(* Logix 5000 project; controller cal1632 1756-L62 rev 16.20; software revision 16.05; part 3 of 57 *)
(* tags used below, declared in another part *)
   AFI : BOOL;
   FAULT : BOOL;
   HMI : BOOL;
   p01_dint_to_hmi : DINT[16];
   p01_param_heater_hl : REAL;
   p01_param_process_air_hl : REAL;
   p01_param_process_air_max : REAL;
   p01_param_temp_limit : REAL;
   p01r01 : routine;
   p01r02 : routine;
   p01r02_all_fans_stopped : BOOL;
   p01r02_batch_run_time : DINT;
   p01r02_batch_run_time_hrs : DINT;
   p01r02_ethernet_comm : DINT;
   p01r02_fault_exists : BOOL;
   p01r02_flash_bit : BOOL;
   p01r02_flash_timer_off : TIMER;
   p01r02_flash_timer_on : TIMER;
   p01r02_plc_faults : DINT;
   p01r02_plc_scan_time : DINT;
   p01r02_plc_scan_time_in_sec : REAL;
   p01r02_timer_batch : TIMER;
   p01r02_timer_fault : TIMER[25];
   p01r02_timer_half_second_off : TIMER;
   p01r02_timer_half_second_on : TIMER;
   p01r02_timer_second : TIMER[2];
   p01r02_timer_warning : TIMER[4];
   p01r02_unack_fault : BOOL;
   p01r02_unack_warning : BOOL;
   p01r02_vfd_comm_2 : DINT[50];
   p01r02_warnings_exists : BOOL;
   p01r03 : routine;
   p01r04 : routine;
   p01r05 : routine;
   p01r06 : routine;
   p01r07 : routine;
   p01r08 : routine;
   p01r09 : routine;
   p01r09_pb_global_reset : BOOL;
   p01r10 : routine;
   p01r11 : routine;
   p01r12 : routine;
   p01r13 : routine;
   p01r13_line_running : BOOL;
   p02_dint_from_hmi : hmi_dint;
   p11r31_request_auto_run : BOOL;
   p11r32_request_auto_run : BOOL;
   p12r31_request_auto_run : BOOL;
   p12r32_request_auto_run : BOOL;
   p13r31_request_auto_run : BOOL;
   p13r32_request_auto_run : BOOL;
   p23_do_enable_impreg_exhaust_fan : BOOL;
   p23r13_request_auto_run : BOOL;

   p26r04_ulb_prs_scp : SYS_SCP := (Input := -85.5, Input_Min := 3.5, Input_Max := 20.0, Output_Min := 5397.0, Output_Max := 30840.0, Output := 5397.0);
   p26r05 : routine := (comment := -1073741761);
   p26r05_timer_fault : TIMER[4];
   p26r05_timer_warning : TIMER[4];
   p26r06 : routine := (comment := -1073741572);
   p26r06_timer_fault : TIMER[4];
   p26r06_timer_warning : TIMER[4];
   p26r07 : routine := (comment := -1073741761);
   p26r07_timer_fault : TIMER[4];
   p26r07_timer_warning : TIMER[4];
   p26r08 : routine := (comment := -1073741761);
   p26r08_timer_fault : TIMER[4];
   p26r08_timer_warning : TIMER[4];
   p26r09 : routine := (comment := -1073741761);
   p26r09_timer_fault : TIMER[4];
   p26r09_timer_warning : TIMER[4];
   p26r10 : routine := (comment := -1073741777);
   p26r10_timer_fault : TIMER[4];
   p26r10_timer_warning : TIMER[4];
   p26r10_ula_selected_tension : REAL := 3.0;
   p26r10_ulb_selected_tension : REAL := 3.0;
   p26r10_unwind_a_brake_torque : REAL := -9.417255;
   p26r10_unwind_a_dia_ft : REAL := -6.2809243;
   p26r10_unwind_b_brake_torque : REAL := -10.6875;
   p26r10_unwind_b_dia_ft : REAL := -7.125;
   p27_ao_dia_a : REAL := -38.8816;
   p27_ao_dia_b : REAL := 8.07605;
   p27_dint_to_hmi : DINT[16] := ([0] := 4);
   p27_inactive_tension_sp : REAL;
   p27_lft_a_prs_input_max : REAL := 30959.0;
   p27_lft_a_prs_input_min : REAL := 200.0;
   p27_lft_a_prs_output_max : REAL := 55.0;
   p27_lft_a_prs_output_min : REAL := 4.0;
   p27_lft_b_prs_input_max : REAL := 30959.0;
   p27_lft_b_prs_input_min : REAL := 60.0;
   p27_lft_b_prs_output_max : REAL := 55.0;
   p27_lft_b_prs_output_min : REAL := 4.0;
   p27_lla_prs_input_max : REAL := 20.0;
   p27_lla_prs_input_min : REAL := 3.5;
   p27_lla_prs_output_max : REAL := 30840.0;
   p27_lla_prs_output_min : REAL := 5397.0;
   p27_lla_prs_scp : SYS_SCP := (Input := -38.914757, Input_Min := 3.5, Input_Max := 20.0, Output_Min := 5397.0, Output_Max := 30840.0, Output := 5397.0);
   p27_llb_prs_input_max : REAL := 20.0;
   p27_llb_prs_input_min : REAL := 3.5;
   p27_llb_prs_output_max : REAL := 30840.0;
   p27_llb_prs_output_min : REAL := 5397.0;
   p27_llb_prs_scp : SYS_SCP := (Input := 8.07605, Input_Min := 3.5, Input_Max := 20.0, Output_Min := 5397.0, Output_Max := 30840.0, Output := 12453.269);
   p27_real_to_hmi : REAL[112] := ([0] := -38.8816, [1] := 8.043039);
   p27r01 : routine := (comment := 7);
   p27r02 : routine := (comment := -1073741761);
   p27r02_fault_exists : BOOL;
   p27r02_timer_fault : TIMER[4];
   p27r02_timer_warning : TIMER[4];
   p27r02_unack_fault : BOOL;
   p27r02_unack_warning : BOOL;
   p27r02_warning_exists : BOOL;
   p27r03 : routine := (comment := -1073741761);
   p27r03_a_radius : REAL := -19.4408;
   p27r03_ai_dia_a_sensor : REAL := 43.9408;
   p27r03_ai_dia_b_sensor : REAL := 8.0619755;
   p27r03_b_radius : REAL := 4.038025;
   p27r03_lower_A_tension_on : BOOL;
   p27r03_lower_B_tension_on : BOOL := 1;
   p27r03_ltf_a_diameter_scp : SYS_SCP := (Input := 24279.0, Input_Min := 200.0, Input_Max := 30959.0, Output_Min := 4.0, Output_Max := 55.0, Output := 43.924217);
   p27r03_ltf_b_diameter_scp : SYS_SCP := (Input := 2521.0, Input_Min := 60.0, Input_Max := 30959.0, Output_Min := 4.0, Output_Max := 55.0, Output := 8.0619755);
   p27r03_timer_fault : TIMER[4];
   p27r03_timer_warning : TIMER[4];
   p27r03_winder_a_distance : REAL := 24.5;
   p27r03_winder_b_distance : REAL := 12.1;
   p27r04 : routine := (comment := -1073741761);
   p27r04_timer_fault : TIMER[4];
   p27r04_timer_warning : TIMER[4];
   p27r05 : routine := (comment := -1073741761);
   p27r05_lla_mode_tension : BOOL;
   p27r05_llb_mode_tension : BOOL := 1;
   p27r05_timer_fault : TIMER[4];
   p27r05_timer_warning : TIMER[4];
   p27r06 : routine := (comment := -1073741572);
   p27r06_timer_fault : TIMER[4];
   p27r06_timer_warning : TIMER[4];
   p27r07 : routine := (comment := -1073741761);
   p27r07_timer_fault : TIMER[4];
   p27r07_timer_warning : TIMER[4];
   p27r08 : routine := (comment := -1073741761);
   p27r08_timer_fault : TIMER[4];
   p27r08_timer_warning : TIMER[4];
   p27r09 : routine := (comment := -1073741761);
   p27r09_a_enable_toggle : SYS_Toggle;
   p27r09_b_enable_toggle : SYS_Toggle := (toggle_state := 1);
   p27r09_timer_fault : TIMER[4];
   p27r09_timer_warning : TIMER[4];
   p27r10 : routine := (comment := -1073741777);
   p27r10_lla_selected_tension : REAL;
   p27r10_llb_selected_tension : REAL := 3.0;
   p27r10_timer_fault : TIMER[4];
   p27r10_timer_warning : TIMER[4];
   p27r10_unwind_a_brake_torque : REAL;
   p27r10_unwind_a_dia_ft : REAL := -3.2428963;
   p27r10_unwind_b_brake_torque : REAL := 1.0095062;
   p27r10_unwind_b_dia_ft : REAL := 0.67300415;
   p27r11 : routine;
   p289_di_ss_jog : BOOL;
   p289_di_ss_run : BOOL;
   p28_ai_slitter_amps : REAL;
   p28_ai_slitter_hz : REAL := -3.8146973e-06;
   p28_ai_slitter_speed : REAL;
   p28_ao_sltr_selected_speed : REAL;
   p28_di_brake : BOOL := 1;
   p28_di_motor : BOOL := 1;
   p28_di_slitter : acs800_di_normal;
   p28_dint_to_hmi : DINT[16] := ([0] := 4, [1] := 1024);
   p28_do_slt_air_supply_sv : BOOL;
   p28_do_sltr : acs800_do_normal;
   p28_real_to_hmi : REAL[112] := ([7] := -3.8146973e-06);
   p28_slitter_on : SYS_Toggle;
   p28r01 : routine := (comment := 7);
   p28r02 : routine := (comment := -1073741761);
   p28r02_fault_exists : BOOL;
   p28r02_timer_fault : TIMER[4];
   p28r02_timer_warning : TIMER[4];
   p28r02_unack_fault : BOOL;
   p28r02_unack_warning : BOOL;
   p28r02_warning_exists : BOOL;
   p28r03 : routine := (comment := -1073741777);
   p28r03_hz : SYS_SCP := (Input_Max := 1800.0, Output_Max := 60.0, Output := -3.8146973e-06);
   p28r03_slitter_speed_fb : SYS_RPM_TO_SPEED := (IN_gear_ratio := 74.24, IN_roll_diameter := 0.5);
   p28r03_timer_fault : TIMER[4];
   p28r03_timer_warning : TIMER[4];
   p28r04 : routine := (comment := -1073741809);
   p28r04_slitter_gear_ratio : REAL := 74.24;
   p28r04_slitter_roll_diameter_ft : REAL := 0.5;
   p28r04_slitter_speed : SYS_SPEED_TO_VFD := (IN_gear_ratio := 74.24, IN_roll_diameter := 0.5);
   p28r04_timer_fault : TIMER[4];
   p28r04_timer_warning : TIMER[4];
   p28r05 : routine := (comment := -1073741809);
   p28r05_timer_fault : TIMER[4];
   p28r05_timer_warning : TIMER[4];
   p28r06 : routine := (comment := -1073741793);
   p28r06_timer_fault : TIMER[4];
   p28r06_timer_warning : TIMER[4];
   p28r07 : routine := (comment := -1073741817);
   p28r07_timer_fault : TIMER[4];
   p28r07_timer_warning : TIMER[4];
   p28r08 : routine := (comment := -1073741769);
   p28r08_timer_fault : TIMER[4];
   p28r08_timer_warning : TIMER[4];
   p28r09 : routine := (comment := -1073741761);
   p28r09_timer_fault : TIMER[4];
   p28r09_timer_warning : TIMER[4];
   p28r10_request_line_run : BOOL;
   p28r11 : routine := (comment := -1073741713, fault := 4, fault_ack := 4);
   p28r11_permissive_run : BOOL;
   p28r11_request_line_jog : BOOL;
   p28r11_request_run : BOOL;
   p28r11_request_thread_fwd : BOOL;
   p28r11_request_thread_rev : BOOL;
   p28r11_slitter_on : BOOL;
   p28r11_timer_fault : TIMER[10] := ([2].ACC := 31, [2].EN := 1, [2].DN := 1);
   p28r11_timer_warning : TIMER[5];
   p29_ai_radius : REAL := 36.375;
   p29_ai_wa_amps : REAL;
   p29_ai_wa_dia_ft : REAL := 0.70011467;
   p29_ai_wa_hz : REAL;
   p29_ai_wa_rpm : REAL;
   p29_ai_wa_speed : REAL;
   p29_ai_wa_torque : REAL;
   p29_ai_wb_amps : REAL;
   p29_ai_wb_dia_ft : REAL := 0.6239968;
   p29_ai_wb_hz : REAL;
   p29_ai_wb_rpm : REAL;
   p29_ai_wb_speed : REAL;
   p29_ai_wb_torque : REAL;
   p29_ai_wdr_dia_in : REAL := 72.75;
   p29_ai_wdr_lc : REAL := 21.484219;
   p29_ai_wdr_turret_amps : REAL;
   p29_ai_wdr_turret_hz : REAL;
   p29_ai_wdr_turret_speed : REAL;
   p29_ao_wa_torque_ref : REAL := 23.650814;
   p29_ao_wb_torque_ref : REAL := 22.166672;
   p29_ao_wda_vfd : REAL;
   p29_ao_wdb_vfd : REAL;
   p29_ao_wdr_turret_selected_speed : REAL;
   p29_ao_wdra_selected_speed : REAL;
   p29_ao_wdrb_selected_speed : REAL;
   p29_di_turret_pos : BOOL := 1;
   p29_di_wa_brake : BOOL := 1;
   p29_di_wa_motor : BOOL := 1;
   p29_di_wb_brake : BOOL := 1;
   p29_di_wb_motor : BOOL := 1;
   p29_di_wdr_a : BOOL := 1;
   p29_di_wdr_a_core_size : BOOL := 1;
   p29_di_wdr_a_reset_core : BOOL;
   p29_di_wdr_a_start : BOOL;
   p29_di_wdr_a_stop : BOOL;
   p29_di_wdr_b_core_size : BOOL := 1;
   p29_di_wdr_b_reset_core : BOOL;
   p29_di_wdr_b_start : BOOL;
   p29_di_wdr_b_stop : BOOL;
   p29_di_wdr_index_fwd : BOOL;
   p29_di_wdr_jog : BOOL;
   p29_di_wdr_turret : acs800_di_normal := (ready := 1, ctrl_from_net := 1, ref_from_net := 1);
   p29_di_wt_motor : BOOL := 1;
   p29_dint_to_hmi : DINT[16] := ([0] := 4, [1] := 4920, [2] := 1285, [3] := 4920, [4] := 512, [5] := 112);
   p29_do_wdr_turret : acs800_do_normal;
   p29_param_fast_turret_speed : REAL := 7.0;
   p29_param_slow_turret_speed : REAL := 5.0;
   p29_param_soak : REAL := 25.0;
   p29_param_wa_gear_ratio : REAL := 50.86;
   p29_param_wb_gear_ratio : REAL := 50.86;
   p29_param_wdt_gear_ratio : REAL := 1200.0;
   p29_param_winder_jog_speed : REAL := 13.0;
   p29_real_to_hmi : REAL[112] := ([0] := 72.75, [1] := 21.454168, [3] := 8.401376, [4] := 7.487962, [21] := 9.277759, [40] := 0.75, [41] := 0.8);
   p29_wa_footage_input_max : REAL := 9000.0;
   p29_wa_footage_input_min : REAL;
   p29_wa_footage_output_max : REAL := 990.0;
   p29_wa_footage_output_min : REAL;
   p29_wb_footage_input_max : REAL := 9000.0;
   p29_wb_footage_input_min : REAL;
   p29_wb_footage_output_max : REAL := 990.0;
   p29_wb_footage_output_min : REAL;
   p29_wda_control_word : INT := 2#0000_0100_0000_0110;
   p29_wda_status_word : INT := 2#0001_0011_0011_1000;
   p29_wda_vfd : ABB_PROTOCOL_VFD := (STATUS_WORD := 4920, CONTROL_WORD := 1030, DRIVE_NOT_READY_FAULT := 1, OUT_FAULT := 1);
   p29_wda_vfd_input_max : REAL := 2000.0;
   p29_wda_vfd_input_min : REAL := -2000.0;
   p29_wda_vfd_output_max : REAL := 20000.0;
   p29_wda_vfd_output_min : REAL := -20000.0;
   p29_wdb_control_word : INT := 2#0000_0100_0000_0110;
   p29_wdb_status_word : INT := 2#0001_0011_0011_1000;
   p29_wdb_vfd : ABB_PROTOCOL_VFD := (STATUS_WORD := 4920, CONTROL_WORD := 1030, DRIVE_NOT_READY_FAULT := 1, OUT_FAULT := 1);
   p29_wdb_vfd_input_max : REAL := 2000.0;
   p29_wdb_vfd_input_min : REAL := -2000.0;
   p29_wdb_vfd_output_max : REAL := 20000.0;
   p29_wdb_vfd_output_min : REAL := -20000.0;
   p29_wdr_diameter_input_max : REAL := 30959.0;
   p29_wdr_diameter_input_min : REAL := 100.0;
   p29_wdr_diameter_output_max : REAL := 55.0;
   p29_wdr_diameter_output_min : REAL := 4.0;
   p29_wdr_lc_input_max : REAL := 10000.0;
   p29_wdr_lc_input_min : REAL;
   p29_wdr_lc_output_max : REAL := 300.0;
   p29_wdr_lc_output_min : REAL;
   p29r01 : routine := (comment := 7);
   p29r02 : routine := (comment := -1073741761);
   p29r02_fault_exists : BOOL := 1;
   p29r02_tension_dev_max : REAL := 85.0;
   p29r02_tension_dev_min : REAL := 55.0;
   p29r02_timer_fault : TIMER[4];
   p29r02_timer_warning : TIMER[4];
   p29r02_unack_fault : BOOL := 1;
   p29r02_unack_warning : BOOL := 1;
   p29r02_wa_calc_torque_ref : REAL := 280.04584;
   p29r02_warning_exists : BOOL := 1;
   p29r02_wb_calc_torque_ref : REAL := 249.59871;
   p29r02_winder_selection_dwell : TIMER := (PRE := 60000, ACC := 60000);
   p29r03 : routine := (comment := -1073741761);
   p29r03_distance_to_core : REAL := 40.375;
   p29r03_hz : SYS_SCP := (Input_Max := 2000.0, Output_Max := 60.0);
   p29r03_liner_wdr_lc_scp : SYS_SCP := (Input := 400.40112, Input_Max := 10000.0, Output_Max := 300.0, Output := 12.012033);
   p29r03_sample_timer : TIMER := (PRE := 200, ACC := 215, EN := 1, DN := 1);
   p29r03_sensor_input : REAL := 4.0;
   p29r03_timer_fault : TIMER[4];
   p29r03_timer_warning : TIMER[4];
   p29r03_unload : REAL;
   p29r03_wa_ave_tq : REAL;
   p29r03_wa_footage_scp : SYS_SCP := (Input := 83.918945, Input_Max := 9000.0, Output_Max := 990.0, Output := 9.231084);
   p29r03_wa_scaled_vfd_in : REAL;
   p29r03_wa_speed_fb : SYS_RPM_TO_SPEED := (IN_gear_ratio := 50.86, IN_roll_diameter := 0.70011467);
   p29r03_wa_tq_ave_ctrl : CONTROL := (LEN := 19);
   p29r03_wa_tq_buffer : REAL[20];
   p29r03_wa_tq_fifo : CONTROL := (LEN := 20, POS := 20, DN := 1);
   p29r03_wb_ave_tq : REAL;
   p29r03_wb_footage_scp : SYS_SCP := (Input := -2.3549805, Input_Max := 9000.0, Output_Max := 990.0);
   p29r03_wb_scaled_vfd_in : REAL;
   p29r03_wb_speed_fb : SYS_RPM_TO_SPEED := (IN_gear_ratio := 50.86, IN_roll_diameter := 0.6239968);
   p29r03_wb_tq_ave_ctrl : CONTROL := (LEN := 19);
   p29r03_wb_tq_buffer : REAL[20];
   p29r03_wb_tq_fifo : CONTROL := (LEN := 20, POS := 20, EN := 1, EU := 1, DN := 1);
   p29r03_wda_vfd_in_scaling : SYS_SCP := (Input_Min := -20000.0, Input_Max := 20000.0, Output_Min := -2000.0, Output_Max := 2000.0);
   p29r03_wda_vfd_input_max : REAL := 20000.0;
   p29r03_wda_vfd_input_min : REAL := -20000.0;
   p29r03_wda_vfd_output_max : REAL := 2000.0;
   p29r03_wda_vfd_output_min : REAL := -2000.0;
   p29r03_wdb_vfd_in_scaling : SYS_SCP := (Input_Min := -20000.0, Input_Max := 20000.0, Output_Min := -2000.0, Output_Max := 2000.0);
   p29r03_wdb_vfd_input_max : REAL := 20000.0;
   p29r03_wdb_vfd_input_min : REAL := -20000.0;
   p29r03_wdb_vfd_output_max : REAL := 2000.0;
   p29r03_wdb_vfd_output_min : REAL := -2000.0;
   p29r03_wdr_dia_sensor_scp : SYS_SCP := (Input_Min := 100.0, Input_Max := 30959.0, Output_Min := 4.0, Output_Max := 55.0, Output := 4.0);
   p29r04 : routine := (comment := -1073741761);
   p29r04_timer_fault : TIMER[4];
   p29r04_timer_warning : TIMER[4];
   p29r04_wda_vfd_out_scaling : SYS_SCP := (Input_Min := -2000.0, Input_Max := 2000.0, Output_Min := -20000.0, Output_Max := 20000.0);
   p29r04_wdb_vfd_out_scaling : SYS_SCP := (Input_Min := -2000.0, Input_Max := 2000.0, Output_Min := -20000.0, Output_Max := 20000.0);
   p29r04_wdr_turret_speed_to_vfd : SYS_SPEED_TO_VFD := (IN_gear_ratio := 1200.0, IN_roll_diameter := 3.2);
   p29r04_wdra_speed_to_vfd : SYS_SPEED_TO_VFD := (IN_gear_ratio := 50.86, IN_roll_diameter := 0.70011467);
   p29r04_wdrb_speed_to_vfd : SYS_SPEED_TO_VFD := (IN_gear_ratio := 50.86, IN_roll_diameter := 0.6239968);
   p29r05 : routine := (comment := -1073741761);
   p29r05_timer_fault : TIMER[4];
   p29r05_timer_warning : TIMER[4];
   p29r06 : routine := (comment := -1073741572);
   p29r06_ave_wdr_lc : REAL := 21.617224;
   p29r06_lc_buffer : REAL[20] := ([0] := 21.441923, [1] := 21.43135, [2] := 21.494793, [3] := 21.37848, [4] := 21.4525, [5] := 21.526514, [6] := 21.526514, [7] := 21.43135, [8] := 21.37848, [9] := 21.441923, [10] := 21.484219, [11] := 21.473642, [12] := 21.558233, [13] := 21.494793, [14] := 21.579384, [15] := 21.537086, [16] := 21.558233, [17] := 21.537086, [18] := 21.537086, [19] := 21.526514);
   p29r06_sample_timer : TIMER := (PRE := 200, ACC := 214, EN := 1, DN := 1);
   p29r06_timer_fault : TIMER[4];
   p29r06_timer_warning : TIMER[4];
   p29r06_unload : REAL := 21.558233;
   p29r06_wdr_lc_ave_ctrl : CONTROL := (LEN := 19);
   p29r06_wdr_lc_fifo : CONTROL := (LEN := 20, POS := 20, DN := 1);
   p29r07 : routine := (comment := -1073741761);
   p29r07_timer_fault : TIMER[4];
   p29r07_timer_warning : TIMER[4];
   p29r08 : routine := (comment := -1073741761);
   p29r08_timer_fault : TIMER[4];
   p29r08_timer_warning : TIMER[4];
   p29r09 : routine := (comment := -1073741761);
   p29r09_ten_ave_len : DINT := 19;
   p29r09_ten_len : DINT := 20;
   p29r09_ten_pos : DINT := 19;
   p29r09_tension_mode : BOOL := 1;
   p29r09_timer_fault : TIMER[4];
   p29r09_timer_warning : TIMER[4];
   p29r09_torque_mode : BOOL;
   p29r09_trq_ave_len : DINT := 999;
   p29r09_trq_len : DINT := 1000;
   p29r09_trq_pos : DINT := 999;
   p29r09_winder_a_active : BOOL := 1;
   p29r09_winder_b_active : BOOL;
   p29r09_winder_jog : BOOL;
   p29r09_winder_off : BOOL := 1;
   p29r09_winder_run : BOOL;
   p29r10 : routine := (comment := -1073740737, oneshot := 2);
   p29r10_accel_bias : REAL := 1.0;
   p29r10_calc_speed_offset : REAL;
   p29r10_index_active : BOOL;
   p29r10_misc_index_factor : REAL := 70.0;
   p29r10_param_psn_gain : REAL := 70.0;
   p29r10_pid_out : REAL := 50.0;
   p29r10_pid_psn : PID := (CTL := -2078244224, EN := 1, SWM := 1, NOBC := 1, INI := 1, DVPA := 1, PVHA := 1, SP := 70.0, KP := 0.75, KI := 0.8, MAXS := 500.0, SO := 50.0, MAXO := 100.0, UPD := 0.01, PV := 21.399628, ERR := 48.600372, OUT := 50.0, MAXI := 500.0, MAXCV := 100.0, MAXTIE := 100.0, DATA[0] := 42.709946, DATA[1] := -68.47881, DATA[2] := 21.399628, DATA[3] := 48.600372, DATA[4] := 70.0, DATA[5] := 0.2, DATA[6] := 1.0, DATA[7] := 0.16, DATA[8] := 0.75, DATA[9] := 0.8, DATA[11] := 0.75, DATA[12] := 0.8, DATA[15] := 1.0, DATA[16] := 1.0);
   p29r10_pid_psn_cv : REAL := 50.0;
   p29r10_pid_psn_pv : REAL := 21.51594;
   p29r10_pid_torque : REAL;
   p29r10_pid_tq : PID := (CTL := -2078244224, EN := 1, SWM := 1, NOBC := 1, INI := 1, DVPA := 1, PVHA := 1, SP := 70.0, KP := 10.0, KI := 0.01, MAXS := 500.0, MAXO := 100.0, UPD := 0.01, PV := 21.420776, ERR := 48.579224, MAXI := 500.0, MAXCV := 80.0, MINCV := 5.0, MAXTIE := 4095.0, DATA[0] := -97.15845, DATA[1] := -68.546486, DATA[2] := 21.420776, DATA[3] := 48.579224, DATA[4] := 70.0, DATA[5] := 0.2, DATA[6] := 1.0, DATA[7] := 0.16, DATA[8] := 10.0, DATA[9] := 0.01, DATA[11] := 10.0, DATA[12] := 0.01, DATA[15] := 0.75, DATA[16] := 0.024420025);
   p29r10_pid_tq_cv : REAL := 5.0;
   p29r10_psn_gain : REAL := 70.0;
   p29r10_request_run : BOOL;
   p29r10_run_permissive : BOOL := 1;
   p29r10_speed_offset : REAL;
   p29r10_timer : TIMER[4] := ([0].PRE := 100, [0].ACC := 122, [0].EN := 1, [0].DN := 1);
   p29r10_timer_fault : TIMER[4];
   p29r10_timer_warning : TIMER[4];
   p29r11 : routine := (comment := -1073740737);
   p29r11_accel_bias : REAL := 1.0;
   p29r11_calc_speed_offset : REAL;
   p29r11_index_active : BOOL;
   p29r11_line_start : BOOL;
   p29r11_line_stop : BOOL;
   p29r11_misc_index_factor : REAL := 70.0;
   p29r11_param_psn_gain : REAL := 70.0;
   p29r11_pid_out : REAL := 50.0;
   p29r11_pid_psn : PID := (CTL := -2078244224, EN := 1, SWM := 1, NOBC := 1, INI := 1, DVPA := 1, PVHA := 1, SP := 70.0, KP := 0.75, KI := 0.8, MAXS := 500.0, SO := 50.0, MAXO := 100.0, UPD := 0.01, PV := 21.399628, ERR := 48.600372, OUT := 50.0, MAXI := 500.0, MAXCV := 100.0, MAXTIE := 100.0, DATA[0] := 42.709946, DATA[1] := -68.47881, DATA[2] := 21.399628, DATA[3] := 48.600372, DATA[4] := 70.0, DATA[5] := 0.2, DATA[6] := 1.0, DATA[7] := 0.16, DATA[8] := 0.75, DATA[9] := 0.8, DATA[11] := 0.75, DATA[12] := 0.8, DATA[15] := 1.0, DATA[16] := 1.0);
   p29r11_pid_psn_cv : REAL := 50.0;
   p29r11_pid_psn_pv : REAL := 21.43135;
   p29r11_pid_torque : REAL := 100.0;
   p29r11_pid_tq : PID := (CTL := -2147446144, EN := 1, INI := 1, OLH := 1, DVPA := 1, PVHA := 1, SP := 70.0, KP := 10.0, KI := 0.01, MAXS := 4095.0, SO := 100.0, MAXO := 100.0, UPD := 0.01, PV := 21.4525, ERR := 48.5475, OUT := 100.0, MAXI := 4095.0, MAXTIE := 4095.0, DATA[0] := 94.45988, DATA[1] := -8.381929, DATA[2] := 21.4525, DATA[3] := 48.5475, DATA[4] := 70.0, DATA[5] := 0.024420025, DATA[6] := 1.0, DATA[7] := 0.16, DATA[8] := 10.0, DATA[9] := 0.01, DATA[11] := 10.0, DATA[12] := 0.01, DATA[16] := 0.024420025);
   p29r11_pid_tq_cv : REAL;
   p29r11_psn_gain : REAL := 70.0;
   p29r11_request_run : BOOL;
   p29r11_run_permissive : BOOL := 1;
   p29r11_speed_offset : REAL;
   p29r11_timer : TIMER[1] := ([0].PRE := 100, [0].ACC := 122, [0].EN := 1, [0].DN := 1);
   p29r11_timer_fault : TIMER[4];
   p29r11_timer_warning : TIMER[4];
   p29r13_ai_wa_footage_ft : REAL := 9.262182;
   p29r13_ai_wb_footage_ft : REAL;
   p29r15 : routine := (comment := -1073741577, fault := 5, unack_fault := 1);
   p29r15_accel_rate : REAL := 25.0;
   p29r15_ao_torque : REAL := 90.0;
   p29r15_const_torque_ref : REAL := 50.0;
   p29r15_decel_rate : REAL := 25.0;
   p29r15_fast_accel_rate : REAL := 25.0;
   p29r15_fast_decel_rate : REAL := 25.0;
   p29r15_index_start_torque : REAL;
   p29r15_jog_torque_ref : REAL := 100.0;
   p29r15_request_jog_fwd : BOOL;
   p29r15_request_run : BOOL;
   p29r15_request_thread_fwd : BOOL;
   p29r15_request_thread_rev : BOOL;
   p29r15_run_permissive : BOOL;
   p29r15_selected_speed : REAL;
   p29r15_selected_torque : REAL := 90.0;
   p29r15_soak_active : BOOL;
   p29r15_state : DINT := 3;
   p29r15_tension_ok : BOOL;
   p29r15_thread_torque_ref : REAL := 100.0;
   p29r15_timer_fault : TIMER[10] := ([0].PRE := 500, [0].ACC := 521, [0].EN := 1, [0].DN := 1, [2].PRE := 2000, [2].ACC := 2021, [2].EN := 1, [2].DN := 1);
   p29r15_timer_warning : TIMER[4] := ([0].PRE := 10000, [1].PRE := 10000, [2].PRE := 10000);
   p29r15_torque_acc_rate : REAL := 0.8;
   p29r15_torque_boost_acc_rate : REAL := 5000.0;
   p29r15_torque_boost_dec_rate : REAL := 2.0;
   p29r15_torque_boost_ref : REAL := 90.0;
   p29r15_torque_boost_timer : TIMER := (PRE := 500);
   p29r15_torque_dec_rate : REAL := 1.6;
   p29r15_torque_fast_acc_rate : REAL := 0.8;
   p29r15_torque_fast_dec_rate : REAL := 1.6;
   p29r15_torque_high_ref : REAL := 100.0;
   p29r15_torque_low_ref : REAL := 1.0;
   p29r15_torque_mode_acc_rate : REAL := 5000.0;
   p29r15_torque_mode_dec_rate : REAL := 4.0;
   p29r15_torque_ramp : SYS_ACC_DEC_RAMP := (IN_selected_line_speed := 90.0, IN_param_master_accel_rate := 0.8, IN_param_master_decel_rate := 1.6, IN_last_scan_s := 0.030536);
   p29r15_torque_soak_acc_rate : REAL := 0.05;
   p29r15_torque_soak_dec_rate : REAL := 0.05;
   p29r15_torque_start_timer : TIMER := (PRE := 200);
   p29r15_wda_vfd_start_request : BOOL;
   p29r15_wdra_accel_decel : SYS_ACC_DEC_RAMP := (IN_param_master_accel_rate := 25.0, IN_param_master_decel_rate := 25.0, IN_last_scan_s := 0.031524);
   p29r15_wdra_active : BOOL;
   p29r15_wdra_ramped_speed : REAL;
   p29r15_zero_speed : BOOL := 1;
   p29r16 : routine := (comment := -1073741577, fault := 5, unack_fault := 1);
   p29r16_accel_rate : REAL := 25.0;
   p29r16_ao_torque : REAL := 90.0;
   p29r16_const_torque_ref : REAL := 50.0;
   p29r16_decel_rate : REAL := 25.0;
   p29r16_fast_accel_rate : REAL := 25.0;
   p29r16_fast_decel_rate : REAL := 25.0;
   p29r16_index_start_torque : REAL;
   p29r16_jog_torque_ref : REAL := 100.0;
   p29r16_request_jog_fwd : BOOL;
   p29r16_request_run : BOOL;
   p29r16_request_thread_fwd : BOOL;
   p29r16_request_thread_rev : BOOL;
   p29r16_run_permissive : BOOL;
   p29r16_selected_speed : REAL;
   p29r16_selected_torque : REAL := 90.0;
   p29r16_soak_active : BOOL;
   p29r16_state : DINT := 3;
   p29r16_tension_ok : BOOL;
   p29r16_thread_torque_ref : REAL := 100.0;
   p29r16_timer_fault : TIMER[10] := ([0].PRE := 500, [0].ACC := 521, [0].EN := 1, [0].DN := 1, [2].PRE := 2000, [2].ACC := 2021, [2].EN := 1, [2].DN := 1);
   p29r16_timer_warning : TIMER[4] := ([0].PRE := 10000, [1].PRE := 10000, [2].PRE := 10000);
   p29r16_torque_acc_rate : REAL := 0.8;
   p29r16_torque_boost_acc_rate : REAL := 5000.0;
   p29r16_torque_boost_dec_rate : REAL := 2.0;
   p29r16_torque_boost_ref : REAL := 90.0;
   p29r16_torque_boost_timer : TIMER := (PRE := 500);
   p29r16_torque_dec_rate : REAL := 1.6;
   p29r16_torque_fast_acc_rate : REAL := 0.8;
   p29r16_torque_fast_dec_rate : REAL := 1.6;
   p29r16_torque_high_ref : REAL := 100.0;
   p29r16_torque_low_ref : REAL := 1.0;
   p29r16_torque_mode_acc_rate : REAL := 5000.0;
   p29r16_torque_mode_dec_rate : REAL := 4.0;
   p29r16_torque_ramp : SYS_ACC_DEC_RAMP := (IN_selected_line_speed := 90.0, IN_param_master_accel_rate := 0.8, IN_param_master_decel_rate := 1.6, IN_last_scan_s := 0.030262);
   p29r16_torque_soak_acc_rate : REAL := 0.05;
   p29r16_torque_soak_dec_rate : REAL := 0.05;
   p29r16_torque_start_timer : TIMER := (PRE := 200);
   p29r16_vfd_start_request : BOOL;
   p29r16_wdrb_accel_decel : SYS_ACC_DEC_RAMP := (IN_param_master_accel_rate := 25.0, IN_param_master_decel_rate := 25.0, IN_last_scan_s := 0.029642);
   p29r16_wdrb_active : BOOL;
   p29r16_wdrb_ramped_speed : REAL;
   p29r16_zero_speed : BOOL := 1;
   p29r17 : routine := (comment := -1073741777);
   p29r17_ave_control : CONTROL := (LEN := 19);
   p29r17_diameter_clac_active : BOOL;
   p29r17_selected_core_diameter : REAL := 6.0;
   p29r17_stack_ctrl : CONTROL := (LEN := 20, POS := 19);
   p29r17_timer : TIMER[5] := ([0].PRE := 20000, [1].PRE := 500);
   p29r17_timer_fault : TIMER[4];
   p29r17_timer_warning : TIMER[4];
   p29r17_winder_a_actual_diam_inch : REAL := 8.367492;
   p29r17_winder_a_avg_diam_inch : REAL := 8.401376;
   p29r17_winder_a_calc_diam_inch : REAL := 8.367492;
   p29r17_winder_a_diam_avg_stack : REAL[1000] := ([0] := 8.476029, [1] := 7.972595, [2] := 8.222083, [3] := 7.8394947, [4] := 8.323315, [5] := 8.169158, [6] := 8.43308, [7] := 8.431416, [8] := 8.535069, [9] := 8.512192, [10] := 9.15567, [11] := 8.434966, [12] := 8.890592, [13] := 8.785833, [14] := 8.268504, [15] := 8.362563, [16] := 8.094648, [17] := 8.356455, [18] := 8.920976, [20] := 6.0, [21] := 6.0, [22] := 6.0, [23] := 6.0, [24] := 6.0, [25] := 6.0, [26] := 6.0, [27] := 6.0, [28] := 6.0, [29] := 6.0, [30] := 6.0, [31] := 6.0, [32] := 6.0, [33] := 6.0, [34] := 6.0, [35] := 6.0, [36] := 6.0, [37] := 6.0, [38] := 6.0, [39] := 6.0, [40] := 6.0, [41] := 6.0, [42] := 6.0, [43] := 6.0, [44] := 6.0, [45] := 6.0, [46] := 6.0, [47] := 6.0, [48] := 6.0, [49] := 6.0, [50] := 6.0, [51] := 6.0, [52] := 6.0, [53] := 6.0, [54] := 6.0, [55] := 6.0, [56] := 6.0, [57] := 6.0, [58] := 6.0, [59] := 6.0, [60] := 6.0,
        [61] := 6.0, [62] := 6.0, [63] := 6.0, [64] := 6.0, [65] := 6.0, [66] := 6.0, [67] := 6.0, [68] := 6.0, [69] := 6.0, [70] := 6.0, [71] := 6.0, [72] := 6.0, [73] := 6.0, [74] := 6.0, [75] := 6.0, [76] := 6.0, [77] := 6.0, [78] := 6.0, [79] := 6.0, [80] := 6.0, [81] := 6.0, [82] := 6.0, [83] := 6.0, [84] := 6.0, [85] := 6.0, [86] := 6.0, [87] := 6.0, [88] := 6.0, [89] := 6.0, [90] := 6.0, [91] := 6.0, [92] := 6.0, [93] := 6.0, [94] := 6.0, [95] := 6.0, [96] := 6.0, [97] := 6.0, [98] := 6.0, [99] := 6.0, [100] := 6.0, [101] := 6.0, [102] := 6.0, [103] := 6.0, [104] := 6.0, [105] := 6.0, [106] := 6.0, [107] := 6.0, [108] := 6.0, [109] := 6.0, [110] := 6.0, [111] := 6.0, [112] := 6.0, [113] := 6.0, [114] := 6.0, [115] := 6.0, [116] := 6.0, [117] := 6.0, [118] := 6.0, [119] := 6.0, [120] := 6.0,
        [121] := 6.0, [122] := 6.0, [123] := 6.0, [124] := 6.0, [125] := 6.0, [126] := 6.0, [127] := 6.0, [128] := 6.0, [129] := 6.0, [130] := 6.0, [131] := 6.0, [132] := 6.0, [133] := 6.0, [134] := 6.0, [135] := 6.0, [136] := 6.0, [137] := 6.0, [138] := 6.0, [139] := 6.0, [140] := 6.0, [141] := 6.0, [142] := 6.0, [143] := 6.0, [144] := 6.0, [145] := 6.0, [146] := 6.0, [147] := 6.0, [148] := 6.0, [149] := 6.0, [150] := 6.0, [151] := 6.0, [152] := 6.0, [153] := 6.0, [154] := 6.0, [155] := 6.0, [156] := 6.0, [157] := 6.0, [158] := 6.0, [159] := 6.0, [160] := 6.0, [161] := 6.0, [162] := 6.0, [163] := 6.0, [164] := 6.0, [165] := 6.0, [166] := 6.0, [167] := 6.0, [168] := 6.0, [169] := 6.0, [170] := 6.0, [171] := 6.0, [172] := 6.0, [173] := 6.0, [174] := 6.0, [175] := 6.0, [176] := 6.0, [177] := 6.0, [178] := 6.0, [179] := 6.0, [180] := 6.0,
        [181] := 6.0, [182] := 6.0, [183] := 6.0, [184] := 6.0, [185] := 6.0, [186] := 6.0, [187] := 6.0, [188] := 6.0, [189] := 6.0, [190] := 6.0, [191] := 6.0, [192] := 6.0, [193] := 6.0, [194] := 6.0, [195] := 6.0, [196] := 6.0, [197] := 6.0, [198] := 6.0, [199] := 6.0, [200] := 6.0, [201] := 6.0, [202] := 6.0, [203] := 6.0, [204] := 6.0, [205] := 6.0, [206] := 6.0, [207] := 6.0, [208] := 6.0, [209] := 6.0, [210] := 6.0, [211] := 6.0, [212] := 6.0, [213] := 6.0, [214] := 6.0, [215] := 6.0, [216] := 6.0, [217] := 6.0, [218] := 6.0, [219] := 6.0, [220] := 6.0, [221] := 6.0, [222] := 6.0, [223] := 6.0, [224] := 6.0, [225] := 6.0, [226] := 6.0, [227] := 6.0, [228] := 6.0, [229] := 6.0, [230] := 6.0, [231] := 6.0, [232] := 6.0, [233] := 6.0, [234] := 6.0, [235] := 6.0, [236] := 6.0, [237] := 6.0, [238] := 6.0, [239] := 6.0, [240] := 6.0,
        [241] := 6.0, [242] := 6.0, [243] := 6.0, [244] := 6.0, [245] := 6.0, [246] := 6.0, [247] := 6.0, [248] := 6.0, [249] := 6.0, [250] := 6.0, [251] := 6.0, [252] := 6.0, [253] := 6.0, [254] := 6.0, [255] := 6.0, [256] := 6.0, [257] := 6.0, [258] := 6.0, [259] := 6.0, [260] := 6.0, [261] := 6.0, [262] := 6.0, [263] := 6.0, [264] := 6.0, [265] := 6.0, [266] := 6.0, [267] := 6.0, [268] := 6.0, [269] := 6.0, [270] := 6.0, [271] := 6.0, [272] := 6.0, [273] := 6.0, [274] := 6.0, [275] := 6.0, [276] := 6.0, [277] := 6.0, [278] := 6.0, [279] := 6.0, [280] := 6.0, [281] := 6.0, [282] := 6.0, [283] := 6.0, [284] := 6.0, [285] := 6.0, [286] := 6.0, [287] := 6.0, [288] := 6.0, [289] := 6.0, [290] := 6.0, [291] := 6.0, [292] := 6.0, [293] := 6.0, [294] := 6.0, [295] := 6.0, [296] := 6.0, [297] := 6.0, [298] := 6.0, [299] := 6.0, [300] := 6.0,
        [301] := 6.0, [302] := 6.0, [303] := 6.0, [304] := 6.0, [305] := 6.0, [306] := 6.0, [307] := 6.0, [308] := 6.0, [309] := 6.0, [310] := 6.0, [311] := 6.0, [312] := 6.0, [313] := 6.0, [314] := 6.0, [315] := 6.0, [316] := 6.0, [317] := 6.0, [318] := 6.0, [319] := 6.0, [320] := 6.0, [321] := 6.0, [322] := 6.0, [323] := 6.0, [324] := 6.0, [325] := 6.0, [326] := 6.0, [327] := 6.0, [328] := 6.0, [329] := 6.0, [330] := 6.0, [331] := 6.0, [332] := 6.0, [333] := 6.0, [334] := 6.0, [335] := 6.0, [336] := 6.0, [337] := 6.0, [338] := 6.0, [339] := 6.0, [340] := 6.0, [341] := 6.0, [342] := 6.0, [343] := 6.0, [344] := 6.0, [345] := 6.0, [346] := 6.0, [347] := 6.0, [348] := 6.0, [349] := 6.0, [350] := 6.0, [351] := 6.0, [352] := 6.0, [353] := 6.0, [354] := 6.0, [355] := 6.0, [356] := 6.0, [357] := 6.0, [358] := 6.0, [359] := 6.0, [360] := 6.0,
        [361] := 6.0, [362] := 6.0, [363] := 6.0, [364] := 6.0, [365] := 6.0, [366] := 6.0, [367] := 6.0, [368] := 6.0, [369] := 6.0, [370] := 6.0, [371] := 6.0, [372] := 6.0, [373] := 6.0, [374] := 6.0, [375] := 6.0, [376] := 6.0, [377] := 6.0, [378] := 6.0, [379] := 6.0, [380] := 6.0, [381] := 6.0, [382] := 6.0, [383] := 6.0, [384] := 6.0, [385] := 6.0, [386] := 6.0, [387] := 6.0, [388] := 6.0, [389] := 6.0, [390] := 6.0, [391] := 6.0, [392] := 6.0, [393] := 6.0, [394] := 6.0, [395] := 6.0, [396] := 6.0, [397] := 6.0, [398] := 6.0, [399] := 6.0, [400] := 6.0, [401] := 6.0, [402] := 6.0, [403] := 6.0, [404] := 6.0, [405] := 6.0, [406] := 6.0, [407] := 6.0, [408] := 6.0, [409] := 6.0, [410] := 6.0, [411] := 6.0, [412] := 6.0, [413] := 6.0, [414] := 6.0, [415] := 6.0, [416] := 6.0, [417] := 6.0, [418] := 6.0, [419] := 6.0, [420] := 6.0,
        [421] := 6.0, [422] := 6.0, [423] := 6.0, [424] := 6.0, [425] := 6.0, [426] := 6.0, [427] := 6.0, [428] := 6.0, [429] := 6.0, [430] := 6.0, [431] := 6.0, [432] := 6.0, [433] := 6.0, [434] := 6.0, [435] := 6.0, [436] := 6.0, [437] := 6.0, [438] := 6.0, [439] := 6.0, [440] := 6.0, [441] := 6.0, [442] := 6.0, [443] := 6.0, [444] := 6.0, [445] := 6.0, [446] := 6.0, [447] := 6.0, [448] := 6.0, [449] := 6.0, [450] := 6.0, [451] := 6.0, [452] := 6.0, [453] := 6.0, [454] := 6.0, [455] := 6.0, [456] := 6.0, [457] := 6.0, [458] := 6.0, [459] := 6.0, [460] := 6.0, [461] := 6.0, [462] := 6.0, [463] := 6.0, [464] := 6.0, [465] := 6.0, [466] := 6.0, [467] := 6.0, [468] := 6.0, [469] := 6.0, [470] := 6.0, [471] := 6.0, [472] := 6.0, [473] := 6.0, [474] := 6.0, [475] := 6.0, [476] := 6.0, [477] := 6.0, [478] := 6.0, [479] := 6.0, [480] := 6.0,
        [481] := 6.0, [482] := 6.0, [483] := 6.0, [484] := 6.0, [485] := 6.0, [486] := 6.0, [487] := 6.0, [488] := 6.0, [489] := 6.0, [490] := 6.0, [491] := 6.0, [492] := 6.0, [493] := 6.0, [494] := 6.0, [495] := 6.0, [496] := 6.0, [497] := 6.0, [498] := 6.0, [499] := 6.0, [500] := 6.0, [501] := 6.0, [502] := 6.0, [503] := 6.0, [504] := 6.0, [505] := 6.0, [506] := 6.0, [507] := 6.0, [508] := 6.0, [509] := 6.0, [510] := 6.0, [511] := 6.0, [512] := 6.0, [513] := 6.0, [514] := 6.0, [515] := 6.0, [516] := 6.0, [517] := 6.0, [518] := 6.0, [519] := 6.0, [520] := 6.0, [521] := 6.0, [522] := 6.0, [523] := 6.0, [524] := 6.0, [525] := 6.0, [526] := 6.0, [527] := 6.0, [528] := 6.0, [529] := 6.0, [530] := 6.0, [531] := 6.0, [532] := 6.0, [533] := 6.0, [534] := 6.0, [535] := 6.0, [536] := 6.0, [537] := 6.0, [538] := 6.0, [539] := 6.0, [540] := 6.0,
        [541] := 6.0, [542] := 6.0, [543] := 6.0, [544] := 6.0, [545] := 6.0, [546] := 6.0, [547] := 6.0, [548] := 6.0, [549] := 6.0, [550] := 6.0, [551] := 6.0, [552] := 6.0, [553] := 6.0, [554] := 6.0, [555] := 6.0, [556] := 6.0, [557] := 6.0, [558] := 6.0, [559] := 6.0, [560] := 6.0, [561] := 6.0, [562] := 6.0, [563] := 6.0, [564] := 6.0, [565] := 6.0, [566] := 6.0, [567] := 6.0, [568] := 6.0, [569] := 6.0, [570] := 6.0, [571] := 6.0, [572] := 6.0, [573] := 6.0, [574] := 6.0, [575] := 6.0, [576] := 6.0, [577] := 6.0, [578] := 6.0, [579] := 6.0, [580] := 6.0, [581] := 6.0, [582] := 6.0, [583] := 6.0, [584] := 6.0, [585] := 6.0, [586] := 6.0, [587] := 6.0, [588] := 6.0, [589] := 6.0, [590] := 6.0, [591] := 6.0, [592] := 6.0, [593] := 6.0, [594] := 6.0, [595] := 6.0, [596] := 6.0, [597] := 6.0, [598] := 6.0, [599] := 6.0, [600] := 6.0,
        [601] := 6.0, [602] := 6.0, [603] := 6.0, [604] := 6.0, [605] := 6.0, [606] := 6.0, [607] := 6.0, [608] := 6.0, [609] := 6.0, [610] := 6.0, [611] := 6.0, [612] := 6.0, [613] := 6.0, [614] := 6.0, [615] := 6.0, [616] := 6.0, [617] := 6.0, [618] := 6.0, [619] := 6.0, [620] := 6.0, [621] := 6.0, [622] := 6.0, [623] := 6.0, [624] := 6.0, [625] := 6.0, [626] := 6.0, [627] := 6.0, [628] := 6.0, [629] := 6.0, [630] := 6.0, [631] := 6.0, [632] := 6.0, [633] := 6.0, [634] := 6.0, [635] := 6.0, [636] := 6.0, [637] := 6.0, [638] := 6.0, [639] := 6.0, [640] := 6.0, [641] := 6.0, [642] := 6.0, [643] := 6.0, [644] := 6.0, [645] := 6.0, [646] := 6.0, [647] := 6.0, [648] := 6.0, [649] := 6.0, [650] := 6.0, [651] := 6.0, [652] := 6.0, [653] := 6.0, [654] := 6.0, [655] := 6.0, [656] := 6.0, [657] := 6.0, [658] := 6.0, [659] := 6.0, [660] := 6.0,
        [661] := 6.0, [662] := 6.0, [663] := 6.0, [664] := 6.0, [665] := 6.0, [666] := 6.0, [667] := 6.0, [668] := 6.0, [669] := 6.0, [670] := 6.0, [671] := 6.0, [672] := 6.0, [673] := 6.0, [674] := 6.0, [675] := 6.0, [676] := 6.0, [677] := 6.0, [678] := 6.0, [679] := 6.0, [680] := 6.0, [681] := 6.0, [682] := 6.0, [683] := 6.0, [684] := 6.0, [685] := 6.0, [686] := 6.0, [687] := 6.0, [688] := 6.0, [689] := 6.0, [690] := 6.0, [691] := 6.0, [692] := 6.0, [693] := 6.0, [694] := 6.0, [695] := 6.0, [696] := 6.0, [697] := 6.0, [698] := 6.0, [699] := 6.0, [700] := 6.0, [701] := 6.0, [702] := 6.0, [703] := 6.0, [704] := 6.0, [705] := 6.0, [706] := 6.0, [707] := 6.0, [708] := 6.0, [709] := 6.0, [710] := 6.0, [711] := 6.0, [712] := 6.0, [713] := 6.0, [714] := 6.0, [715] := 6.0, [716] := 6.0, [717] := 6.0, [718] := 6.0, [719] := 6.0, [720] := 6.0,
        [721] := 6.0, [722] := 6.0, [723] := 6.0, [724] := 6.0, [725] := 6.0, [726] := 6.0, [727] := 6.0, [728] := 6.0, [729] := 6.0, [730] := 6.0, [731] := 6.0, [732] := 6.0, [733] := 6.0, [734] := 6.0, [735] := 6.0, [736] := 6.0, [737] := 6.0, [738] := 6.0, [739] := 6.0, [740] := 6.0, [741] := 6.0, [742] := 6.0, [743] := 6.0, [744] := 6.0, [745] := 6.0, [746] := 6.0, [747] := 6.0, [748] := 6.0, [749] := 6.0, [750] := 6.0, [751] := 6.0, [752] := 6.0, [753] := 6.0, [754] := 6.0, [755] := 6.0, [756] := 6.0, [757] := 6.0, [758] := 6.0, [759] := 6.0, [760] := 6.0, [761] := 6.0, [762] := 6.0, [763] := 6.0, [764] := 6.0, [765] := 6.0, [766] := 6.0, [767] := 6.0, [768] := 6.0, [769] := 6.0, [770] := 6.0, [771] := 6.0, [772] := 6.0, [773] := 6.0, [774] := 6.0, [775] := 6.0, [776] := 6.0, [777] := 6.0, [778] := 6.0, [779] := 6.0, [780] := 6.0,
        [781] := 6.0, [782] := 6.0, [783] := 6.0, [784] := 6.0, [785] := 6.0, [786] := 6.0, [787] := 6.0, [788] := 6.0, [789] := 6.0, [790] := 6.0, [791] := 6.0, [792] := 6.0, [793] := 6.0, [794] := 6.0, [795] := 6.0, [796] := 6.0, [797] := 6.0, [798] := 6.0, [799] := 6.0, [800] := 6.0, [801] := 6.0, [802] := 6.0, [803] := 6.0, [804] := 6.0, [805] := 6.0, [806] := 6.0, [807] := 6.0, [808] := 6.0, [809] := 6.0, [810] := 6.0, [811] := 6.0, [812] := 6.0, [813] := 6.0, [814] := 6.0, [815] := 6.0, [816] := 6.0, [817] := 6.0, [818] := 6.0, [819] := 6.0, [820] := 6.0, [821] := 6.0, [822] := 6.0, [823] := 6.0, [824] := 6.0, [825] := 6.0, [826] := 6.0, [827] := 6.0, [828] := 6.0, [829] := 6.0, [830] := 6.0, [831] := 6.0, [832] := 6.0, [833] := 6.0, [834] := 6.0, [835] := 6.0, [836] := 6.0, [837] := 6.0, [838] := 6.0, [839] := 6.0, [840] := 6.0,
        [841] := 6.0, [842] := 6.0, [843] := 6.0, [844] := 6.0, [845] := 6.0, [846] := 6.0, [847] := 6.0, [848] := 6.0, [849] := 6.0, [850] := 6.0, [851] := 6.0, [852] := 6.0, [853] := 6.0, [854] := 6.0, [855] := 6.0, [856] := 6.0, [857] := 6.0, [858] := 6.0, [859] := 6.0, [860] := 6.0, [861] := 6.0, [862] := 6.0, [863] := 6.0, [864] := 6.0, [865] := 6.0, [866] := 6.0, [867] := 6.0, [868] := 6.0, [869] := 6.0, [870] := 6.0, [871] := 6.0, [872] := 6.0, [873] := 6.0, [874] := 6.0, [875] := 6.0, [876] := 6.0, [877] := 6.0, [878] := 6.0, [879] := 6.0, [880] := 6.0, [881] := 6.0, [882] := 6.0, [883] := 6.0, [884] := 6.0, [885] := 6.0, [886] := 6.0, [887] := 6.0, [888] := 6.0, [889] := 6.0, [890] := 6.0, [891] := 6.0, [892] := 6.0, [893] := 6.0, [894] := 6.0, [895] := 6.0, [896] := 6.0, [897] := 6.0, [898] := 6.0, [899] := 6.0, [900] := 6.0,
        [901] := 6.0, [902] := 6.0, [903] := 6.0, [904] := 6.0, [905] := 6.0, [906] := 6.0, [907] := 6.0, [908] := 6.0, [909] := 6.0, [910] := 6.0, [911] := 6.0, [912] := 6.0, [913] := 6.0, [914] := 6.0, [915] := 6.0, [916] := 6.0, [917] := 6.0, [918] := 6.0, [919] := 6.0, [920] := 6.0, [921] := 6.0, [922] := 6.0, [923] := 6.0, [924] := 6.0, [925] := 6.0, [926] := 6.0, [927] := 6.0, [928] := 6.0, [929] := 6.0, [930] := 6.0, [931] := 6.0, [932] := 6.0, [933] := 6.0, [934] := 6.0, [935] := 6.0, [936] := 6.0, [937] := 6.0, [938] := 6.0, [939] := 6.0, [940] := 6.0, [941] := 6.0, [942] := 6.0, [943] := 6.0, [944] := 6.0, [945] := 6.0, [946] := 6.0, [947] := 6.0, [948] := 6.0, [949] := 6.0, [950] := 6.0, [951] := 6.0, [952] := 6.0, [953] := 6.0, [954] := 6.0, [955] := 6.0, [956] := 6.0, [957] := 6.0, [958] := 6.0, [959] := 6.0, [960] := 6.0,
        [961] := 6.0, [962] := 6.0, [963] := 6.0, [964] := 6.0, [965] := 6.0, [966] := 6.0, [967] := 6.0, [968] := 6.0, [969] := 6.0, [970] := 6.0, [971] := 6.0, [972] := 6.0, [973] := 6.0, [974] := 6.0, [975] := 6.0, [976] := 6.0, [977] := 6.0, [978] := 6.0, [979] := 6.0, [980] := 6.0, [981] := 6.0, [982] := 6.0, [983] := 6.0, [984] := 6.0, [985] := 6.0, [986] := 6.0, [987] := 6.0, [988] := 6.0, [989] := 6.0, [990] := 6.0, [991] := 6.0, [992] := 6.0, [993] := 6.0, [994] := 6.0, [995] := 6.0, [996] := 6.0, [997] := 6.0, [998] := 6.0, [999] := 6.0);
   p29r17_winder_a_selected_diam_inch : REAL := 6.0;
   p29r17_winder_a_unload : REAL := 8.362458;
   p29r18 : routine := (comment := -1073741777);
   p29r18_ave_control : CONTROL := (LEN := 19);
   p29r18_diameter_calc_active : BOOL;
   p29r18_min_tension : REAL := 10.0;
   p29r18_selected_core_diameter : REAL := 6.0;
   p29r18_stack_ctrl : CONTROL := (LEN := 20, POS := 19);
   p29r18_timer : TIMER[5] := ([0].PRE := 20000, [1].PRE := 500);
   p29r18_timer_fault : TIMER[4];
   p29r18_timer_warning : TIMER[4];
   p29r18_winder_b_actual_diam_inch : REAL := 7.32814;
   p29r18_winder_b_avg_diam_inch : REAL := 7.487962;
   p29r18_winder_b_calc_diam_inch : REAL := 7.32814;
   p29r18_winder_b_diam_avg_stack : REAL[1000] := ([0] := 7.6374273, [1] := 7.610406, [2] := 7.2743893, [3] := 7.3928, [4] := 7.38477, [5] := 7.6354856, [6] := 7.303881, [7] := 7.6925106, [8] := 7.445376, [9] := 7.2835655, [10] := 7.5873795, [11] := 7.613444, [12] := 7.405342, [13] := 7.5007663, [14] := 7.682413, [15] := 7.560098, [16] := 7.3233614, [17] := 7.5467844, [18] := 7.2874413, [20] := 6.0, [21] := 6.0, [22] := 6.0, [23] := 6.0, [24] := 6.0, [25] := 6.0, [26] := 6.0, [27] := 6.0, [28] := 6.0, [29] := 6.0, [30] := 6.0, [31] := 6.0, [32] := 6.0, [33] := 6.0, [34] := 6.0, [35] := 6.0, [36] := 6.0, [37] := 6.0, [38] := 6.0, [39] := 6.0, [40] := 6.0, [41] := 6.0, [42] := 6.0, [43] := 6.0, [44] := 6.0, [45] := 6.0, [46] := 6.0, [47] := 6.0, [48] := 6.0, [49] := 6.0, [50] := 6.0, [51] := 6.0, [52] := 6.0, [53] := 6.0, [54] := 6.0, [55] := 6.0, [56] := 6.0, [57] := 6.0, [58] := 6.0, [59] := 6.0, [60] := 6.0,
        [61] := 6.0, [62] := 6.0, [63] := 6.0, [64] := 6.0, [65] := 6.0, [66] := 6.0, [67] := 6.0, [68] := 6.0, [69] := 6.0, [70] := 6.0, [71] := 6.0, [72] := 6.0, [73] := 6.0, [74] := 6.0, [75] := 6.0, [76] := 6.0, [77] := 6.0, [78] := 6.0, [79] := 6.0, [80] := 6.0, [81] := 6.0, [82] := 6.0, [83] := 6.0, [84] := 6.0, [85] := 6.0, [86] := 6.0, [87] := 6.0, [88] := 6.0, [89] := 6.0, [90] := 6.0, [91] := 6.0, [92] := 6.0, [93] := 6.0, [94] := 6.0, [95] := 6.0, [96] := 6.0, [97] := 6.0, [98] := 6.0, [99] := 6.0, [100] := 6.0, [101] := 6.0, [102] := 6.0, [103] := 6.0, [104] := 6.0, [105] := 6.0, [106] := 6.0, [107] := 6.0, [108] := 6.0, [109] := 6.0, [110] := 6.0, [111] := 6.0, [112] := 6.0, [113] := 6.0, [114] := 6.0, [115] := 6.0, [116] := 6.0, [117] := 6.0, [118] := 6.0, [119] := 6.0, [120] := 6.0,
        [121] := 6.0, [122] := 6.0, [123] := 6.0, [124] := 6.0, [125] := 6.0, [126] := 6.0, [127] := 6.0, [128] := 6.0, [129] := 6.0, [130] := 6.0, [131] := 6.0, [132] := 6.0, [133] := 6.0, [134] := 6.0, [135] := 6.0, [136] := 6.0, [137] := 6.0, [138] := 6.0, [139] := 6.0, [140] := 6.0, [141] := 6.0, [142] := 6.0, [143] := 6.0, [144] := 6.0, [145] := 6.0, [146] := 6.0, [147] := 6.0, [148] := 6.0, [149] := 6.0, [150] := 6.0, [151] := 6.0, [152] := 6.0, [153] := 6.0, [154] := 6.0, [155] := 6.0, [156] := 6.0, [157] := 6.0, [158] := 6.0, [159] := 6.0, [160] := 6.0, [161] := 6.0, [162] := 6.0, [163] := 6.0, [164] := 6.0, [165] := 6.0, [166] := 6.0, [167] := 6.0, [168] := 6.0, [169] := 6.0, [170] := 6.0, [171] := 6.0, [172] := 6.0, [173] := 6.0, [174] := 6.0, [175] := 6.0, [176] := 6.0, [177] := 6.0, [178] := 6.0, [179] := 6.0, [180] := 6.0,
        [181] := 6.0, [182] := 6.0, [183] := 6.0, [184] := 6.0, [185] := 6.0, [186] := 6.0, [187] := 6.0, [188] := 6.0, [189] := 6.0, [190] := 6.0, [191] := 6.0, [192] := 6.0, [193] := 6.0, [194] := 6.0, [195] := 6.0, [196] := 6.0, [197] := 6.0, [198] := 6.0, [199] := 6.0, [200] := 6.0, [201] := 6.0, [202] := 6.0, [203] := 6.0, [204] := 6.0, [205] := 6.0, [206] := 6.0, [207] := 6.0, [208] := 6.0, [209] := 6.0, [210] := 6.0, [211] := 6.0, [212] := 6.0, [213] := 6.0, [214] := 6.0, [215] := 6.0, [216] := 6.0, [217] := 6.0, [218] := 6.0, [219] := 6.0, [220] := 6.0, [221] := 6.0, [222] := 6.0, [223] := 6.0, [224] := 6.0, [225] := 6.0, [226] := 6.0, [227] := 6.0, [228] := 6.0, [229] := 6.0, [230] := 6.0, [231] := 6.0, [232] := 6.0, [233] := 6.0, [234] := 6.0, [235] := 6.0, [236] := 6.0, [237] := 6.0, [238] := 6.0, [239] := 6.0, [240] := 6.0,
        [241] := 6.0, [242] := 6.0, [243] := 6.0, [244] := 6.0, [245] := 6.0, [246] := 6.0, [247] := 6.0, [248] := 6.0, [249] := 6.0, [250] := 6.0, [251] := 6.0, [252] := 6.0, [253] := 6.0, [254] := 6.0, [255] := 6.0, [256] := 6.0, [257] := 6.0, [258] := 6.0, [259] := 6.0, [260] := 6.0, [261] := 6.0, [262] := 6.0, [263] := 6.0, [264] := 6.0, [265] := 6.0, [266] := 6.0, [267] := 6.0, [268] := 6.0, [269] := 6.0, [270] := 6.0, [271] := 6.0, [272] := 6.0, [273] := 6.0, [274] := 6.0, [275] := 6.0, [276] := 6.0, [277] := 6.0, [278] := 6.0, [279] := 6.0, [280] := 6.0, [281] := 6.0, [282] := 6.0, [283] := 6.0, [284] := 6.0, [285] := 6.0, [286] := 6.0, [287] := 6.0, [288] := 6.0, [289] := 6.0, [290] := 6.0, [291] := 6.0, [292] := 6.0, [293] := 6.0, [294] := 6.0, [295] := 6.0, [296] := 6.0, [297] := 6.0, [298] := 6.0, [299] := 6.0, [300] := 6.0,
        [301] := 6.0, [302] := 6.0, [303] := 6.0, [304] := 6.0, [305] := 6.0, [306] := 6.0, [307] := 6.0, [308] := 6.0, [309] := 6.0, [310] := 6.0, [311] := 6.0, [312] := 6.0, [313] := 6.0, [314] := 6.0, [315] := 6.0, [316] := 6.0, [317] := 6.0, [318] := 6.0, [319] := 6.0, [320] := 6.0, [321] := 6.0, [322] := 6.0, [323] := 6.0, [324] := 6.0, [325] := 6.0, [326] := 6.0, [327] := 6.0, [328] := 6.0, [329] := 6.0, [330] := 6.0, [331] := 6.0, [332] := 6.0, [333] := 6.0, [334] := 6.0, [335] := 6.0, [336] := 6.0, [337] := 6.0, [338] := 6.0, [339] := 6.0, [340] := 6.0, [341] := 6.0, [342] := 6.0, [343] := 6.0, [344] := 6.0, [345] := 6.0, [346] := 6.0, [347] := 6.0, [348] := 6.0, [349] := 6.0, [350] := 6.0, [351] := 6.0, [352] := 6.0, [353] := 6.0, [354] := 6.0, [355] := 6.0, [356] := 6.0, [357] := 6.0, [358] := 6.0, [359] := 6.0, [360] := 6.0,
        [361] := 6.0, [362] := 6.0, [363] := 6.0, [364] := 6.0, [365] := 6.0, [366] := 6.0, [367] := 6.0, [368] := 6.0, [369] := 6.0, [370] := 6.0, [371] := 6.0, [372] := 6.0, [373] := 6.0, [374] := 6.0, [375] := 6.0, [376] := 6.0, [377] := 6.0, [378] := 6.0, [379] := 6.0, [380] := 6.0, [381] := 6.0, [382] := 6.0, [383] := 6.0, [384] := 6.0, [385] := 6.0, [386] := 6.0, [387] := 6.0, [388] := 6.0, [389] := 6.0, [390] := 6.0, [391] := 6.0, [392] := 6.0, [393] := 6.0, [394] := 6.0, [395] := 6.0, [396] := 6.0, [397] := 6.0, [398] := 6.0, [399] := 6.0, [400] := 6.0, [401] := 6.0, [402] := 6.0, [403] := 6.0, [404] := 6.0, [405] := 6.0, [406] := 6.0, [407] := 6.0, [408] := 6.0, [409] := 6.0, [410] := 6.0, [411] := 6.0, [412] := 6.0, [413] := 6.0, [414] := 6.0, [415] := 6.0, [416] := 6.0, [417] := 6.0, [418] := 6.0, [419] := 6.0, [420] := 6.0,
        [421] := 6.0, [422] := 6.0, [423] := 6.0, [424] := 6.0, [425] := 6.0, [426] := 6.0, [427] := 6.0, [428] := 6.0, [429] := 6.0, [430] := 6.0, [431] := 6.0, [432] := 6.0, [433] := 6.0, [434] := 6.0, [435] := 6.0, [436] := 6.0, [437] := 6.0, [438] := 6.0, [439] := 6.0, [440] := 6.0, [441] := 6.0, [442] := 6.0, [443] := 6.0, [444] := 6.0, [445] := 6.0, [446] := 6.0, [447] := 6.0, [448] := 6.0, [449] := 6.0, [450] := 6.0, [451] := 6.0, [452] := 6.0, [453] := 6.0, [454] := 6.0, [455] := 6.0, [456] := 6.0, [457] := 6.0, [458] := 6.0, [459] := 6.0, [460] := 6.0, [461] := 6.0, [462] := 6.0, [463] := 6.0, [464] := 6.0, [465] := 6.0, [466] := 6.0, [467] := 6.0, [468] := 6.0, [469] := 6.0, [470] := 6.0, [471] := 6.0, [472] := 6.0, [473] := 6.0, [474] := 6.0, [475] := 6.0, [476] := 6.0, [477] := 6.0, [478] := 6.0, [479] := 6.0, [480] := 6.0,
        [481] := 6.0, [482] := 6.0, [483] := 6.0, [484] := 6.0, [485] := 6.0, [486] := 6.0, [487] := 6.0, [488] := 6.0, [489] := 6.0, [490] := 6.0, [491] := 6.0, [492] := 6.0, [493] := 6.0, [494] := 6.0, [495] := 6.0, [496] := 6.0, [497] := 6.0, [498] := 6.0, [499] := 6.0, [500] := 6.0, [501] := 6.0, [502] := 6.0, [503] := 6.0, [504] := 6.0, [505] := 6.0, [506] := 6.0, [507] := 6.0, [508] := 6.0, [509] := 6.0, [510] := 6.0, [511] := 6.0, [512] := 6.0, [513] := 6.0, [514] := 6.0, [515] := 6.0, [516] := 6.0, [517] := 6.0, [518] := 6.0, [519] := 6.0, [520] := 6.0, [521] := 6.0, [522] := 6.0, [523] := 6.0, [524] := 6.0, [525] := 6.0, [526] := 6.0, [527] := 6.0, [528] := 6.0, [529] := 6.0, [530] := 6.0, [531] := 6.0, [532] := 6.0, [533] := 6.0, [534] := 6.0, [535] := 6.0, [536] := 6.0, [537] := 6.0, [538] := 6.0, [539] := 6.0, [540] := 6.0,
        [541] := 6.0, [542] := 6.0, [543] := 6.0, [544] := 6.0, [545] := 6.0, [546] := 6.0, [547] := 6.0, [548] := 6.0, [549] := 6.0, [550] := 6.0, [551] := 6.0, [552] := 6.0, [553] := 6.0, [554] := 6.0, [555] := 6.0, [556] := 6.0, [557] := 6.0, [558] := 6.0, [559] := 6.0, [560] := 6.0, [561] := 6.0, [562] := 6.0, [563] := 6.0, [564] := 6.0, [565] := 6.0, [566] := 6.0, [567] := 6.0, [568] := 6.0, [569] := 6.0, [570] := 6.0, [571] := 6.0, [572] := 6.0, [573] := 6.0, [574] := 6.0, [575] := 6.0, [576] := 6.0, [577] := 6.0, [578] := 6.0, [579] := 6.0, [580] := 6.0, [581] := 6.0, [582] := 6.0, [583] := 6.0, [584] := 6.0, [585] := 6.0, [586] := 6.0, [587] := 6.0, [588] := 6.0, [589] := 6.0, [590] := 6.0, [591] := 6.0, [592] := 6.0, [593] := 6.0, [594] := 6.0, [595] := 6.0, [596] := 6.0, [597] := 6.0, [598] := 6.0, [599] := 6.0, [600] := 6.0,
        [601] := 6.0, [602] := 6.0, [603] := 6.0, [604] := 6.0, [605] := 6.0, [606] := 6.0, [607] := 6.0, [608] := 6.0, [609] := 6.0, [610] := 6.0, [611] := 6.0, [612] := 6.0, [613] := 6.0, [614] := 6.0, [615] := 6.0, [616] := 6.0, [617] := 6.0, [618] := 6.0, [619] := 6.0, [620] := 6.0, [621] := 6.0, [622] := 6.0, [623] := 6.0, [624] := 6.0, [625] := 6.0, [626] := 6.0, [627] := 6.0, [628] := 6.0, [629] := 6.0, [630] := 6.0, [631] := 6.0, [632] := 6.0, [633] := 6.0, [634] := 6.0, [635] := 6.0, [636] := 6.0, [637] := 6.0, [638] := 6.0, [639] := 6.0, [640] := 6.0, [641] := 6.0, [642] := 6.0, [643] := 6.0, [644] := 6.0, [645] := 6.0, [646] := 6.0, [647] := 6.0, [648] := 6.0, [649] := 6.0, [650] := 6.0, [651] := 6.0, [652] := 6.0, [653] := 6.0, [654] := 6.0, [655] := 6.0, [656] := 6.0, [657] := 6.0, [658] := 6.0, [659] := 6.0, [660] := 6.0,
        [661] := 6.0, [662] := 6.0, [663] := 6.0, [664] := 6.0, [665] := 6.0, [666] := 6.0, [667] := 6.0, [668] := 6.0, [669] := 6.0, [670] := 6.0, [671] := 6.0, [672] := 6.0, [673] := 6.0, [674] := 6.0, [675] := 6.0, [676] := 6.0, [677] := 6.0, [678] := 6.0, [679] := 6.0, [680] := 6.0, [681] := 6.0, [682] := 6.0, [683] := 6.0, [684] := 6.0, [685] := 6.0, [686] := 6.0, [687] := 6.0, [688] := 6.0, [689] := 6.0, [690] := 6.0, [691] := 6.0, [692] := 6.0, [693] := 6.0, [694] := 6.0, [695] := 6.0, [696] := 6.0, [697] := 6.0, [698] := 6.0, [699] := 6.0, [700] := 6.0, [701] := 6.0, [702] := 6.0, [703] := 6.0, [704] := 6.0, [705] := 6.0, [706] := 6.0, [707] := 6.0, [708] := 6.0, [709] := 6.0, [710] := 6.0, [711] := 6.0, [712] := 6.0, [713] := 6.0, [714] := 6.0, [715] := 6.0, [716] := 6.0, [717] := 6.0, [718] := 6.0, [719] := 6.0, [720] := 6.0,
        [721] := 6.0, [722] := 6.0, [723] := 6.0, [724] := 6.0, [725] := 6.0, [726] := 6.0, [727] := 6.0, [728] := 6.0, [729] := 6.0, [730] := 6.0, [731] := 6.0, [732] := 6.0, [733] := 6.0, [734] := 6.0, [735] := 6.0, [736] := 6.0, [737] := 6.0, [738] := 6.0, [739] := 6.0, [740] := 6.0, [741] := 6.0, [742] := 6.0, [743] := 6.0, [744] := 6.0, [745] := 6.0, [746] := 6.0, [747] := 6.0, [748] := 6.0, [749] := 6.0, [750] := 6.0, [751] := 6.0, [752] := 6.0, [753] := 6.0, [754] := 6.0, [755] := 6.0, [756] := 6.0, [757] := 6.0, [758] := 6.0, [759] := 6.0, [760] := 6.0, [761] := 6.0, [762] := 6.0, [763] := 6.0, [764] := 6.0, [765] := 6.0, [766] := 6.0, [767] := 6.0, [768] := 6.0, [769] := 6.0, [770] := 6.0, [771] := 6.0, [772] := 6.0, [773] := 6.0, [774] := 6.0, [775] := 6.0, [776] := 6.0, [777] := 6.0, [778] := 6.0, [779] := 6.0, [780] := 6.0,
        [781] := 6.0, [782] := 6.0, [783] := 6.0, [784] := 6.0, [785] := 6.0, [786] := 6.0, [787] := 6.0, [788] := 6.0, [789] := 6.0, [790] := 6.0, [791] := 6.0, [792] := 6.0, [793] := 6.0, [794] := 6.0, [795] := 6.0, [796] := 6.0, [797] := 6.0, [798] := 6.0, [799] := 6.0, [800] := 6.0, [801] := 6.0, [802] := 6.0, [803] := 6.0, [804] := 6.0, [805] := 6.0, [806] := 6.0, [807] := 6.0, [808] := 6.0, [809] := 6.0, [810] := 6.0, [811] := 6.0, [812] := 6.0, [813] := 6.0, [814] := 6.0, [815] := 6.0, [816] := 6.0, [817] := 6.0, [818] := 6.0, [819] := 6.0, [820] := 6.0, [821] := 6.0, [822] := 6.0, [823] := 6.0, [824] := 6.0, [825] := 6.0, [826] := 6.0, [827] := 6.0, [828] := 6.0, [829] := 6.0, [830] := 6.0, [831] := 6.0, [832] := 6.0, [833] := 6.0, [834] := 6.0, [835] := 6.0, [836] := 6.0, [837] := 6.0, [838] := 6.0, [839] := 6.0, [840] := 6.0,
        [841] := 6.0, [842] := 6.0, [843] := 6.0, [844] := 6.0, [845] := 6.0, [846] := 6.0, [847] := 6.0, [848] := 6.0, [849] := 6.0, [850] := 6.0, [851] := 6.0, [852] := 6.0, [853] := 6.0, [854] := 6.0, [855] := 6.0, [856] := 6.0, [857] := 6.0, [858] := 6.0, [859] := 6.0, [860] := 6.0, [861] := 6.0, [862] := 6.0, [863] := 6.0, [864] := 6.0, [865] := 6.0, [866] := 6.0, [867] := 6.0, [868] := 6.0, [869] := 6.0, [870] := 6.0, [871] := 6.0, [872] := 6.0, [873] := 6.0, [874] := 6.0, [875] := 6.0, [876] := 6.0, [877] := 6.0, [878] := 6.0, [879] := 6.0, [880] := 6.0, [881] := 6.0, [882] := 6.0, [883] := 6.0, [884] := 6.0, [885] := 6.0, [886] := 6.0, [887] := 6.0, [888] := 6.0, [889] := 6.0, [890] := 6.0, [891] := 6.0, [892] := 6.0, [893] := 6.0, [894] := 6.0, [895] := 6.0, [896] := 6.0, [897] := 6.0, [898] := 6.0, [899] := 6.0, [900] := 6.0,
        [901] := 6.0, [902] := 6.0, [903] := 6.0, [904] := 6.0, [905] := 6.0, [906] := 6.0, [907] := 6.0, [908] := 6.0, [909] := 6.0, [910] := 6.0, [911] := 6.0, [912] := 6.0, [913] := 6.0, [914] := 6.0, [915] := 6.0, [916] := 6.0, [917] := 6.0, [918] := 6.0, [919] := 6.0, [920] := 6.0, [921] := 6.0, [922] := 6.0, [923] := 6.0, [924] := 6.0, [925] := 6.0, [926] := 6.0, [927] := 6.0, [928] := 6.0, [929] := 6.0, [930] := 6.0, [931] := 6.0, [932] := 6.0, [933] := 6.0, [934] := 6.0, [935] := 6.0, [936] := 6.0, [937] := 6.0, [938] := 6.0, [939] := 6.0, [940] := 6.0, [941] := 6.0, [942] := 6.0, [943] := 6.0, [944] := 6.0, [945] := 6.0, [946] := 6.0, [947] := 6.0, [948] := 6.0, [949] := 6.0, [950] := 6.0, [951] := 6.0, [952] := 6.0, [953] := 6.0, [954] := 6.0, [955] := 6.0, [956] := 6.0, [957] := 6.0, [958] := 6.0, [959] := 6.0, [960] := 6.0,
        [961] := 6.0, [962] := 6.0, [963] := 6.0, [964] := 6.0, [965] := 6.0, [966] := 6.0, [967] := 6.0, [968] := 6.0, [969] := 6.0, [970] := 6.0, [971] := 6.0, [972] := 6.0, [973] := 6.0, [974] := 6.0, [975] := 6.0, [976] := 6.0, [977] := 6.0, [978] := 6.0, [979] := 6.0, [980] := 6.0, [981] := 6.0, [982] := 6.0, [983] := 6.0, [984] := 6.0, [985] := 6.0, [986] := 6.0, [987] := 6.0, [988] := 6.0, [989] := 6.0, [990] := 6.0, [991] := 6.0, [992] := 6.0, [993] := 6.0, [994] := 6.0, [995] := 6.0, [996] := 6.0, [997] := 6.0, [998] := 6.0, [999] := 6.0);
   p29r18_winder_b_selected_diam_inch : REAL := 6.0;
   p29r18_winder_b_unload : REAL := 7.3910923;
   p29r20 : routine := (comment := -1073738505, warning := 2, unack_warning := 1, state := 3);
   p29r20_acc_dec_ramp : SYS_ACC_DEC_RAMP := (IN_param_master_accel_rate := 2.0, IN_param_master_decel_rate := 2.0, IN_last_scan_s := 0.030346);
   p29r20_accel_rate : REAL := 2.0;
   p29r20_decel_rate : REAL := 2.0;
   p29r20_fast_accel : REAL := 2.0;
   p29r20_fast_decel : REAL := 2.0;
   p29r20_index_complete : BOOL := 1;
   p29r20_index_move_timer : TIMER;
   p29r20_permissive : BOOL := 1;
   p29r20_request_fwd : BOOL;
   p29r20_request_rev : BOOL;
   p29r20_selected_speed : REAL;
   p29r20_timer_fault : TIMER[10];
   p29r20_timer_warning : TIMER[4] := ([1].ACC := 32, [1].EN := 1, [1].DN := 1);
   p29r20_zero_speed : BOOL := 1;
   p30_di_pin_1 : BOOL := 1;
   p30_di_pin_2 : BOOL := 1;
   p30_di_pin_3 : BOOL := 1;
   p30_di_pin_4 : BOOL := 1;
   p30_di_pin_5 : BOOL := 1;
   p30_di_pin_6 : BOOL := 1;
   p30_di_pin_7 : BOOL := 1;
   p30_di_pin_8 : BOOL := 1;
   p30_di_retraction_down_ls : BOOL := 1;
   p30_di_retraction_up_ls : BOOL;
   p30_di_rotation_fault : BOOL;
   p30_di_ss_close : BOOL;
   p30_di_ss_open : BOOL;
   p30_dint_to_hmi : DINT[16] := ([0] := 255);
   p30_do_retract_motion : BOOL;
   p30_do_rotation_fwd : BOOL;
   p30_do_rotation_rev : BOOL;
   p30_real_to_hmi : REAL[112];
   p30r01 : routine := (comment := 7);
   p30r02 : routine := (comment := -1073741761);
   p30r02_fault_exists : BOOL;
   p30r02_timer_fault : TIMER[4];
   p30r02_timer_warning : TIMER[4];
   p30r02_unack_fault : BOOL;
   p30r02_unack_warning : BOOL;
   p30r02_warning_exists : BOOL;
   p30r03 : routine := (comment := -1073741761);
   p30r03_timer_fault : TIMER[4];
   p30r03_timer_warning : TIMER[4];
   p30r04 : routine := (comment := -1073741761);
   p30r04_timer_fault : TIMER[4];
   p30r04_timer_warning : TIMER[4];
   p30r05 : routine := (comment := -1073741761);
   p30r05_timer_fault : TIMER[4];
   p30r05_timer_warning : TIMER[4];
   p30r06 : routine := (comment := -1073741572);
   p30r06_timer_fault : TIMER[4];
   p30r06_timer_warning : TIMER[4];
   p30r07 : routine := (comment := -1073741761);
   p30r07_timer_fault : TIMER[4];
   p30r07_timer_warning : TIMER[4];
   p30r08 : routine := (comment := -1073741761);
   p30r08_timer_fault : TIMER[4];
   p30r08_timer_warning : TIMER[4];
   p30r09 : routine := (comment := -1073741761);
   p30r09_mode_close : BOOL;
   p30r09_mode_off : BOOL := 1;
   p30r09_mode_open : BOOL;
   p30r09_timer_fault : TIMER[4];
   p30r09_timer_warning : TIMER[4];
   p30r10 : routine := (comment := -1073741777);
   p30r10_motion_monitor_dwell : TIMER := (PRE := 500);
   p30r10_request_close : BOOL;
   p30r10_request_monitor : BOOL;
   p30r10_request_open : BOOL;
   p30r10_run_permissive : BOOL := 1;
   p30r10_safety_pins_stowed : BOOL := 1;
   p30r10_state : DINT;
   p30r10_timer_fault : TIMER[4] := ([0].PRE := 500, [1].PRE := 400);
   p30r10_timer_warning : TIMER[4] := ([0].PRE := 1000);
   p31r09 : routine;
   p32r13_request_auto_stop : BOOL;
   poo_vfd_sprng_HMI_hand : BOOL;
   RETACTION_DELAY_TIMER : TIMER := (PRE := 4000);
   RETRACTION_DELAY_TIMER_2 : TIMER := (PRE := 4000);
   spd_vfd_jog_tmr : TIMER := (PRE := 30000);
   spring_spd_adj_prcnt : REAL := 0.98;
END_VAR

PROGRAM P01_System   (* main routine R01_Main *)

ROUTINE R01_Main   (* ladder *)
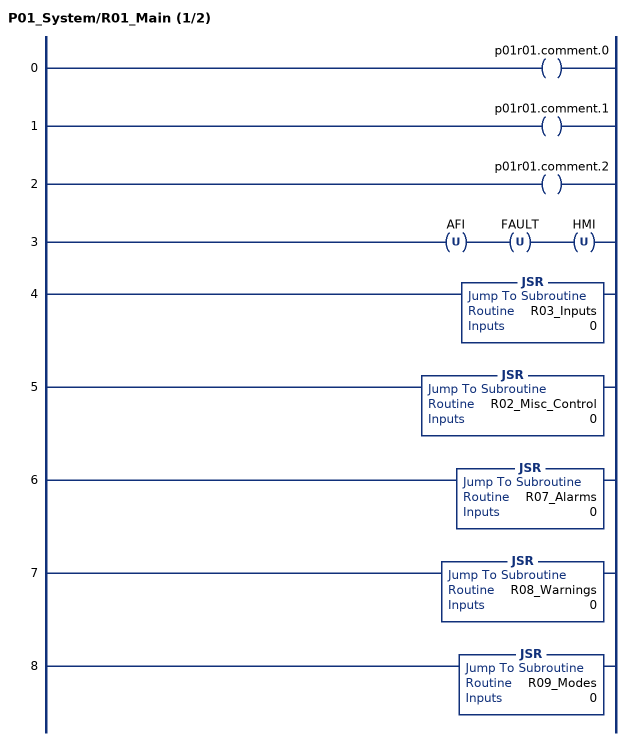
   0: OTE(p01r01.comment.0);
   1: OTE(p01r01.comment.1);
   2: OTE(p01r01.comment.2);
   3: OTU(AFI)OTU(FAULT)OTU(HMI);
   4: JSR(R03_Inputs,0);
   5: JSR(R02_Misc_Control,0);
   6: JSR(R07_Alarms,0);
   7: JSR(R08_Warnings,0);
   8: JSR(R09_Modes,0);
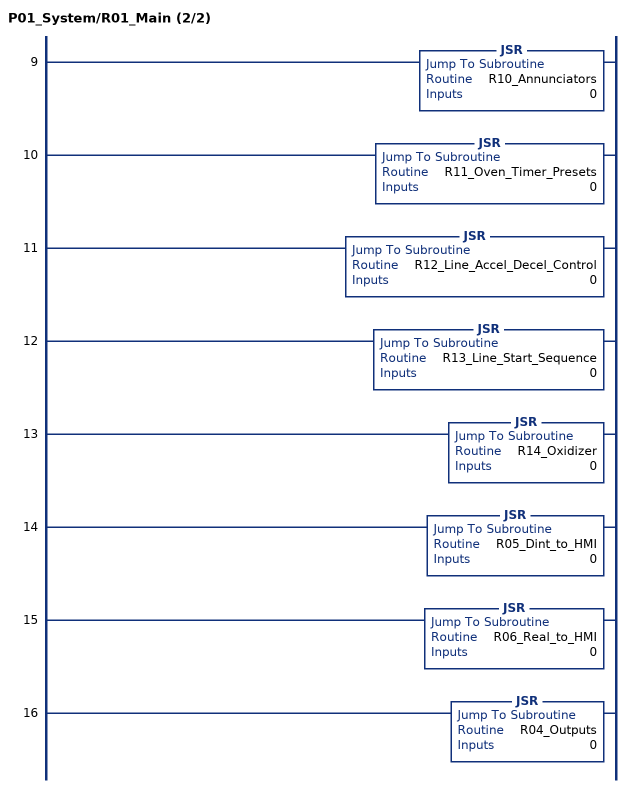
   9: JSR(R10_Annunciators,0);
   10: JSR(R11_Oven_Timer_Presets,0);
   11: JSR(R12_Line_Accel_Decel_Control,0);
   12: JSR(R13_Line_Start_Sequence,0);
   13: JSR(R14_Oxidizer,0);
   14: JSR(R05_Dint_to_HMI,0);
   15: JSR(R06_Real_to_HMI,0);
   16: JSR(R04_Outputs,0);
END_ROUTINE

ROUTINE R02_Misc_Control   (* ladder *)
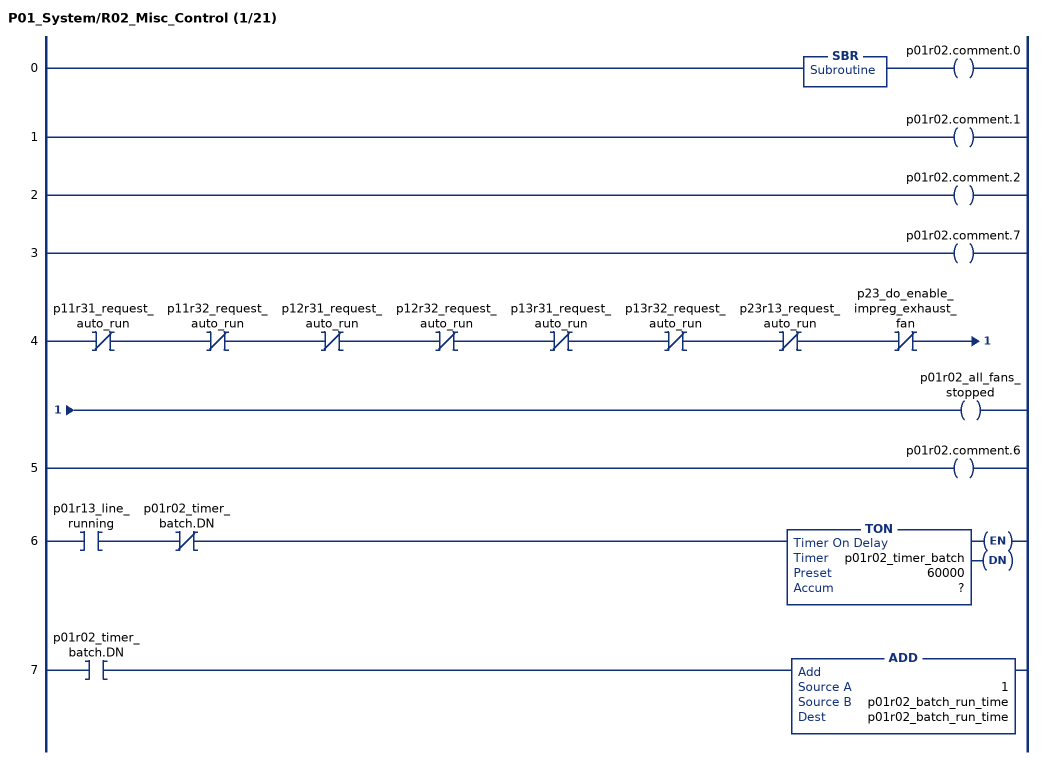
   0: SBR()OTE(p01r02.comment.0);
   1: OTE(p01r02.comment.1);
   2: OTE(p01r02.comment.2);
   3: OTE(p01r02.comment.7);
   4: XIO(p11r31_request_auto_run)XIO(p11r32_request_auto_run)XIO(p12r31_request_auto_run)XIO(p12r32_request_auto_run)XIO(p13r31_request_auto_run)XIO(p13r32_request_auto_run)XIO(p23r13_request_auto_run)XIO(p23_do_enable_impreg_exhaust_fan)OTE(p01r02_all_fans_stopped);
   5: OTE(p01r02.comment.6);
   6: XIC(p01r13_line_running)XIO(p01r02_timer_batch.DN)TON(p01r02_timer_batch,?,?);
   7: XIC(p01r02_timer_batch.DN)ADD(1,p01r02_batch_run_time,p01r02_batch_run_time);
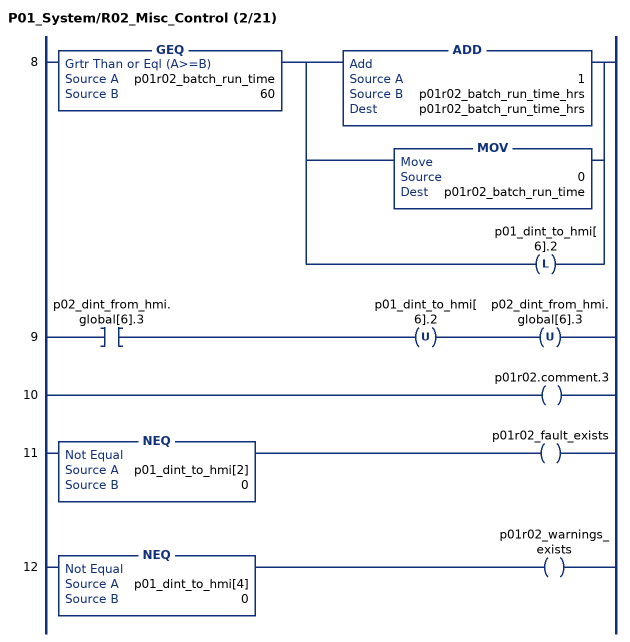
   8: GEQ(p01r02_batch_run_time,60)[ADD(1,p01r02_batch_run_time_hrs,p01r02_batch_run_time_hrs) ,MOV(0,p01r02_batch_run_time) ,OTL(p01_dint_to_hmi[6].2) ];
   9: XIC(p02_dint_from_hmi.global[6].3)OTU(p01_dint_to_hmi[6].2)OTU(p02_dint_from_hmi.global[6].3);
   10: OTE(p01r02.comment.3);
   11: NEQ(p01_dint_to_hmi[2],0)OTE(p01r02_fault_exists);
   12: NEQ(p01_dint_to_hmi[4],0)OTE(p01r02_warnings_exists);
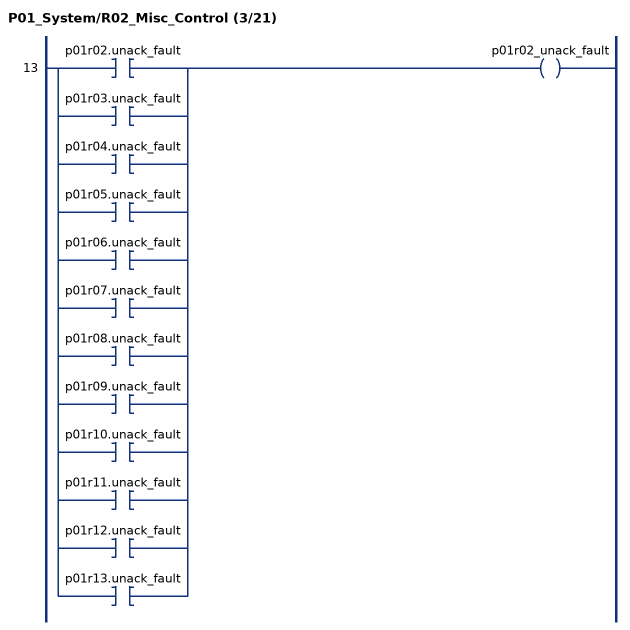
   13: [XIC(p01r02.unack_fault) ,XIC(p01r03.unack_fault) ,XIC(p01r04.unack_fault) ,XIC(p01r05.unack_fault) ,XIC(p01r06.unack_fault) ,XIC(p01r07.unack_fault) ,XIC(p01r08.unack_fault) ,XIC(p01r09.unack_fault) ,XIC(p01r10.unack_fault) ,XIC(p01r11.unack_fault) ,XIC(p01r12.unack_fault) ,XIC(p01r13.unack_fault) ]OTE(p01r02_unack_fault);
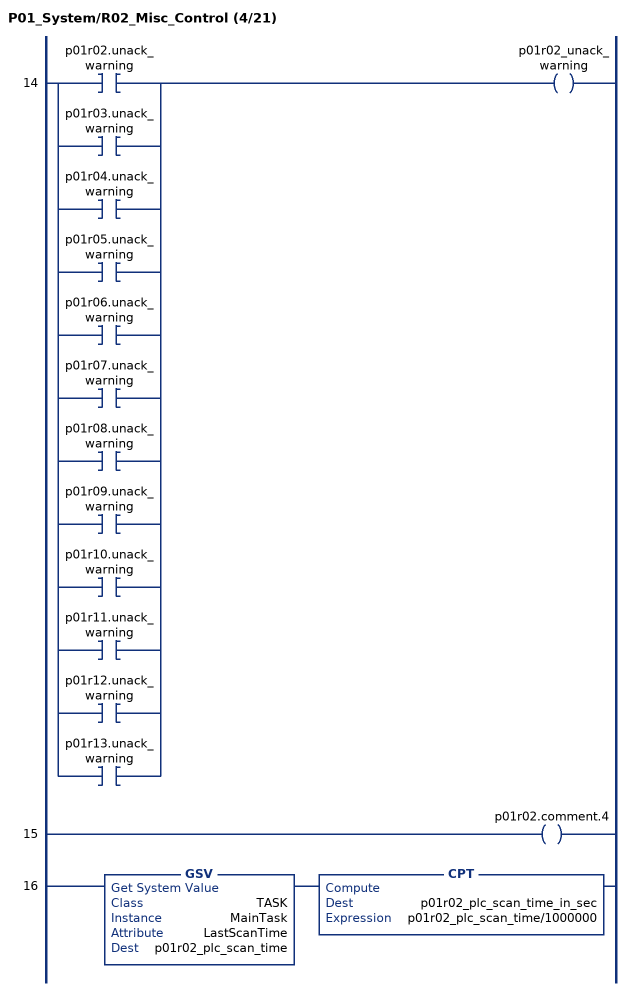
   14: [XIC(p01r02.unack_warning) ,XIC(p01r03.unack_warning) ,XIC(p01r04.unack_warning) ,XIC(p01r05.unack_warning) ,XIC(p01r06.unack_warning) ,XIC(p01r07.unack_warning) ,XIC(p01r08.unack_warning) ,XIC(p01r09.unack_warning) ,XIC(p01r10.unack_warning) ,XIC(p01r11.unack_warning) ,XIC(p01r12.unack_warning) ,XIC(p01r13.unack_warning) ]OTE(p01r02_unack_warning);
   15: OTE(p01r02.comment.4);
   16: GSV(TASK,MainTask,LastScanTime,p01r02_plc_scan_time)CPT(p01r02_plc_scan_time_in_sec,p01r02_plc_scan_time/1000000);
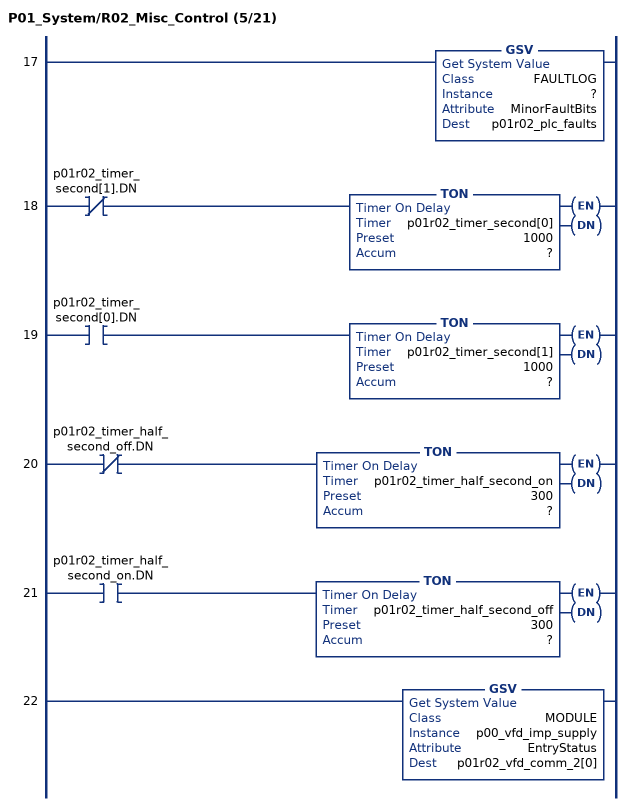
   17: GSV(FAULTLOG,?,MinorFaultBits,p01r02_plc_faults);
   18: XIO(p01r02_timer_second[1].DN)TON(p01r02_timer_second[0],?,?);
   19: XIC(p01r02_timer_second[0].DN)TON(p01r02_timer_second[1],?,?);
   20: XIO(p01r02_timer_half_second_off.DN)TON(p01r02_timer_half_second_on,?,?);
   21: XIC(p01r02_timer_half_second_on.DN)TON(p01r02_timer_half_second_off,?,?);
   22: GSV(MODULE,p00_vfd_imp_supply,EntryStatus,p01r02_vfd_comm_2[0]);
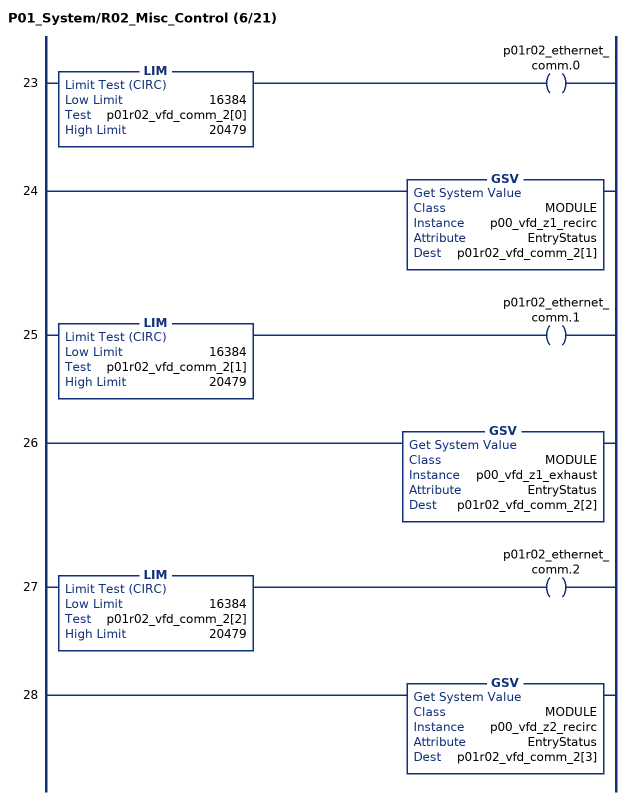
   23: LIM(16384,p01r02_vfd_comm_2[0],20479)OTE(p01r02_ethernet_comm.0);
   24: GSV(MODULE,p00_vfd_z1_recirc,EntryStatus,p01r02_vfd_comm_2[1]);
   25: LIM(16384,p01r02_vfd_comm_2[1],20479)OTE(p01r02_ethernet_comm.1);
   26: GSV(MODULE,p00_vfd_z1_exhaust,EntryStatus,p01r02_vfd_comm_2[2]);
   27: LIM(16384,p01r02_vfd_comm_2[2],20479)OTE(p01r02_ethernet_comm.2);
   28: GSV(MODULE,p00_vfd_z2_recirc,EntryStatus,p01r02_vfd_comm_2[3]);
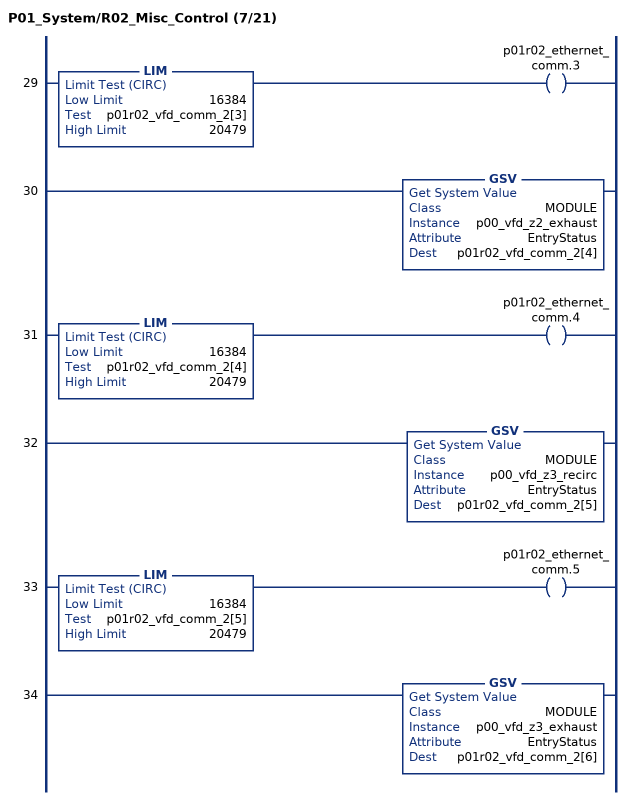
   29: LIM(16384,p01r02_vfd_comm_2[3],20479)OTE(p01r02_ethernet_comm.3);
   30: GSV(MODULE,p00_vfd_z2_exhaust,EntryStatus,p01r02_vfd_comm_2[4]);
   31: LIM(16384,p01r02_vfd_comm_2[4],20479)OTE(p01r02_ethernet_comm.4);
   32: GSV(MODULE,p00_vfd_z3_recirc,EntryStatus,p01r02_vfd_comm_2[5]);
   33: LIM(16384,p01r02_vfd_comm_2[5],20479)OTE(p01r02_ethernet_comm.5);
   34: GSV(MODULE,p00_vfd_z3_exhaust,EntryStatus,p01r02_vfd_comm_2[6]);
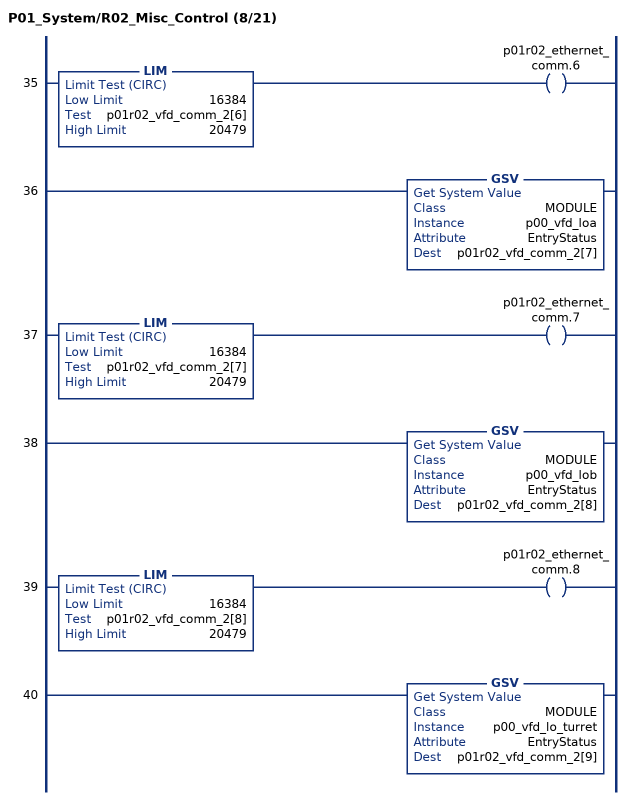
   35: LIM(16384,p01r02_vfd_comm_2[6],20479)OTE(p01r02_ethernet_comm.6);
   36: GSV(MODULE,p00_vfd_loa,EntryStatus,p01r02_vfd_comm_2[7]);
   37: LIM(16384,p01r02_vfd_comm_2[7],20479)OTE(p01r02_ethernet_comm.7);
   38: GSV(MODULE,p00_vfd_lob,EntryStatus,p01r02_vfd_comm_2[8]);
   39: LIM(16384,p01r02_vfd_comm_2[8],20479)OTE(p01r02_ethernet_comm.8);
   40: GSV(MODULE,p00_vfd_lo_turret,EntryStatus,p01r02_vfd_comm_2[9]);
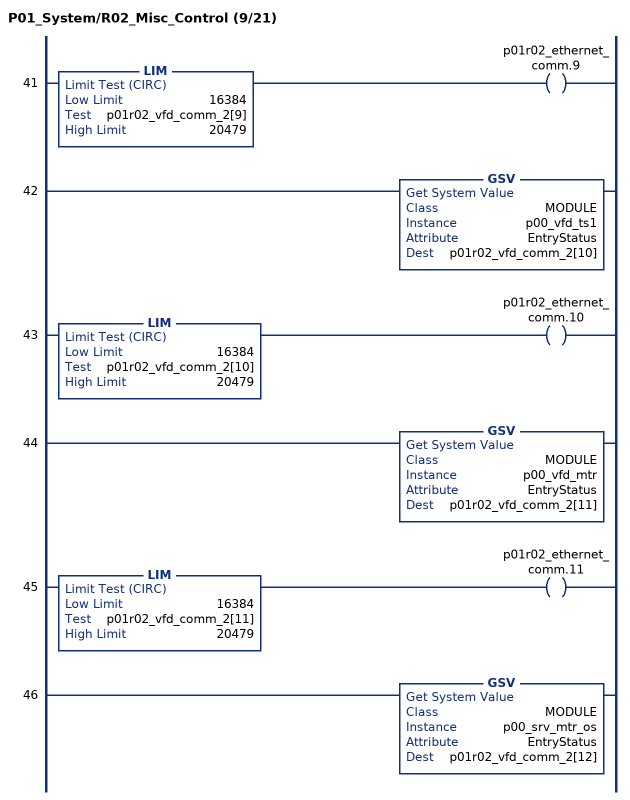
   41: LIM(16384,p01r02_vfd_comm_2[9],20479)OTE(p01r02_ethernet_comm.9);
   42: GSV(MODULE,p00_vfd_ts1,EntryStatus,p01r02_vfd_comm_2[10]);
   43: LIM(16384,p01r02_vfd_comm_2[10],20479)OTE(p01r02_ethernet_comm.10);
   44: GSV(MODULE,p00_vfd_mtr,EntryStatus,p01r02_vfd_comm_2[11]);
   45: LIM(16384,p01r02_vfd_comm_2[11],20479)OTE(p01r02_ethernet_comm.11);
   46: GSV(MODULE,p00_srv_mtr_os,EntryStatus,p01r02_vfd_comm_2[12]);
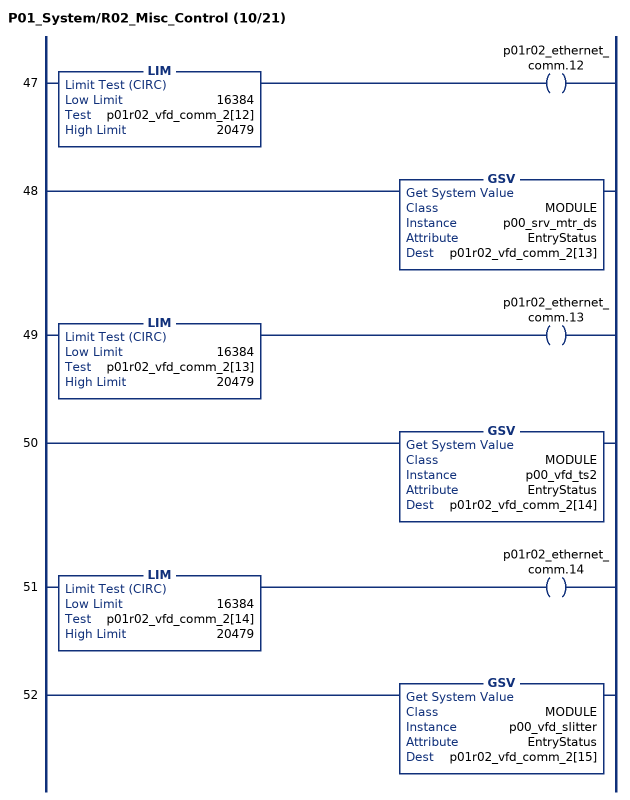
   47: LIM(16384,p01r02_vfd_comm_2[12],20479)OTE(p01r02_ethernet_comm.12);
   48: GSV(MODULE,p00_srv_mtr_ds,EntryStatus,p01r02_vfd_comm_2[13]);
   49: LIM(16384,p01r02_vfd_comm_2[13],20479)OTE(p01r02_ethernet_comm.13);
   50: GSV(MODULE,p00_vfd_ts2,EntryStatus,p01r02_vfd_comm_2[14]);
   51: LIM(16384,p01r02_vfd_comm_2[14],20479)OTE(p01r02_ethernet_comm.14);
   52: GSV(MODULE,p00_vfd_slitter,EntryStatus,p01r02_vfd_comm_2[15]);
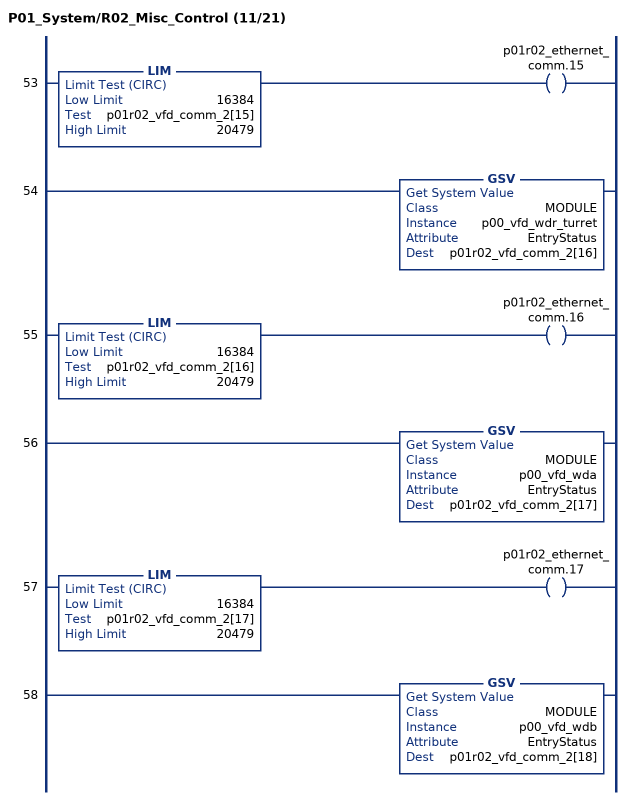
   53: LIM(16384,p01r02_vfd_comm_2[15],20479)OTE(p01r02_ethernet_comm.15);
   54: GSV(MODULE,p00_vfd_wdr_turret,EntryStatus,p01r02_vfd_comm_2[16]);
   55: LIM(16384,p01r02_vfd_comm_2[16],20479)OTE(p01r02_ethernet_comm.16);
   56: GSV(MODULE,p00_vfd_wda,EntryStatus,p01r02_vfd_comm_2[17]);
   57: LIM(16384,p01r02_vfd_comm_2[17],20479)OTE(p01r02_ethernet_comm.17);
   58: GSV(MODULE,p00_vfd_wdb,EntryStatus,p01r02_vfd_comm_2[18]);
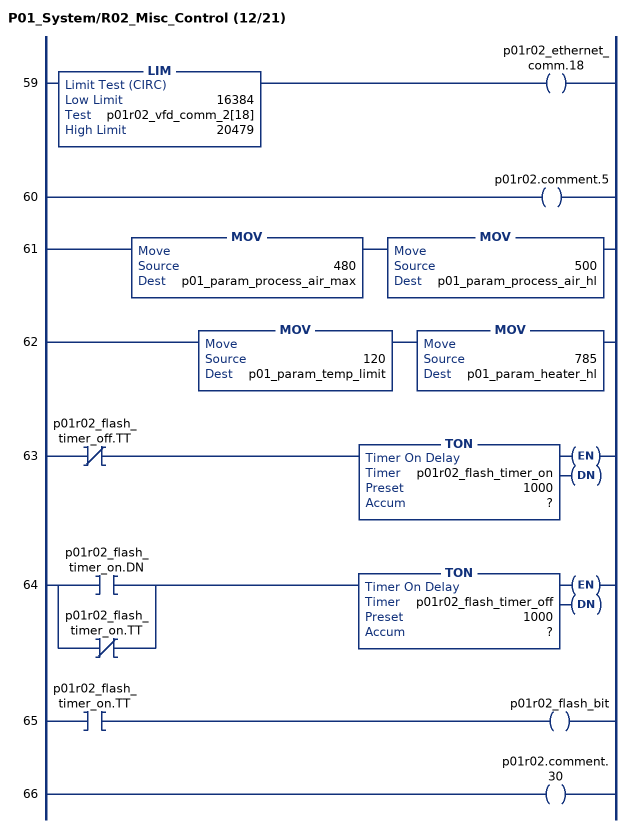
   59: LIM(16384,p01r02_vfd_comm_2[18],20479)OTE(p01r02_ethernet_comm.18);
   60: OTE(p01r02.comment.5);
   61: MOV(480,p01_param_process_air_max)MOV(500,p01_param_process_air_hl);
   62: MOV(120,p01_param_temp_limit)MOV(785,p01_param_heater_hl);
   63: XIO(p01r02_flash_timer_off.TT)TON(p01r02_flash_timer_on,?,?);
   64: [XIC(p01r02_flash_timer_on.DN) ,XIO(p01r02_flash_timer_on.TT) ]TON(p01r02_flash_timer_off,?,?);
   65: XIC(p01r02_flash_timer_on.TT)OTE(p01r02_flash_bit);
   66: OTE(p01r02.comment.30);
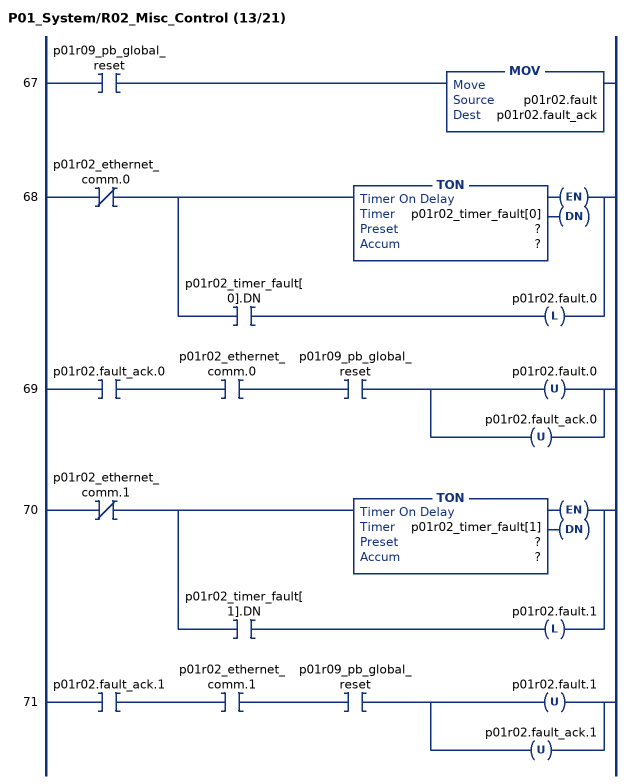
   67: XIC(p01r09_pb_global_reset)MOV(p01r02.fault,p01r02.fault_ack);
   68: XIO(p01r02_ethernet_comm.0)[TON(p01r02_timer_fault[0],?,?) ,XIC(p01r02_timer_fault[0].DN) OTL(p01r02.fault.0) ];
   69: XIC(p01r02.fault_ack.0)XIC(p01r02_ethernet_comm.0)XIC(p01r09_pb_global_reset)[OTU(p01r02.fault.0) ,OTU(p01r02.fault_ack.0) ];
   70: XIO(p01r02_ethernet_comm.1)[TON(p01r02_timer_fault[1],?,?) ,XIC(p01r02_timer_fault[1].DN) OTL(p01r02.fault.1) ];
   71: XIC(p01r02.fault_ack.1)XIC(p01r02_ethernet_comm.1)XIC(p01r09_pb_global_reset)[OTU(p01r02.fault.1) ,OTU(p01r02.fault_ack.1) ];
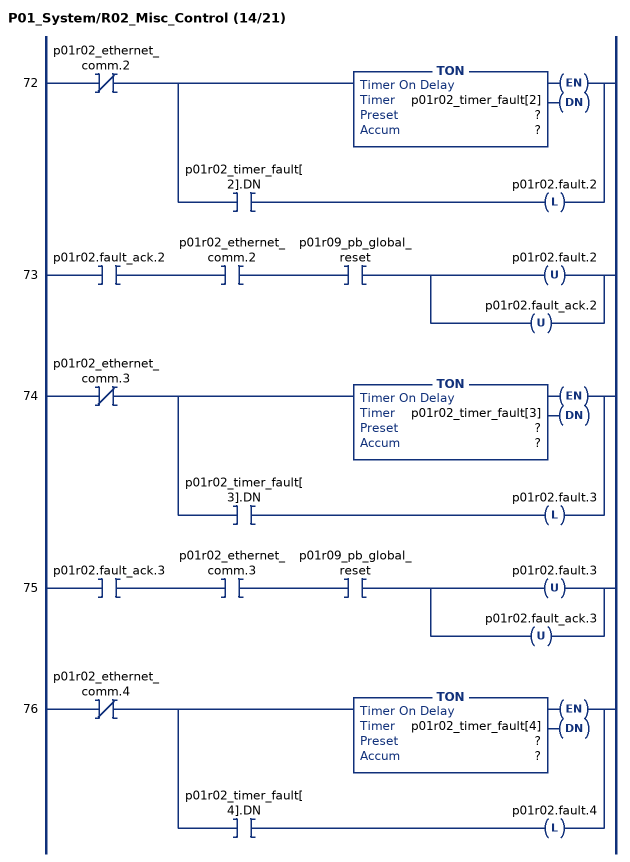
   72: XIO(p01r02_ethernet_comm.2)[TON(p01r02_timer_fault[2],?,?) ,XIC(p01r02_timer_fault[2].DN) OTL(p01r02.fault.2) ];
   73: XIC(p01r02.fault_ack.2)XIC(p01r02_ethernet_comm.2)XIC(p01r09_pb_global_reset)[OTU(p01r02.fault.2) ,OTU(p01r02.fault_ack.2) ];
   74: XIO(p01r02_ethernet_comm.3)[TON(p01r02_timer_fault[3],?,?) ,XIC(p01r02_timer_fault[3].DN) OTL(p01r02.fault.3) ];
   75: XIC(p01r02.fault_ack.3)XIC(p01r02_ethernet_comm.3)XIC(p01r09_pb_global_reset)[OTU(p01r02.fault.3) ,OTU(p01r02.fault_ack.3) ];
   76: XIO(p01r02_ethernet_comm.4)[TON(p01r02_timer_fault[4],?,?) ,XIC(p01r02_timer_fault[4].DN) OTL(p01r02.fault.4) ];
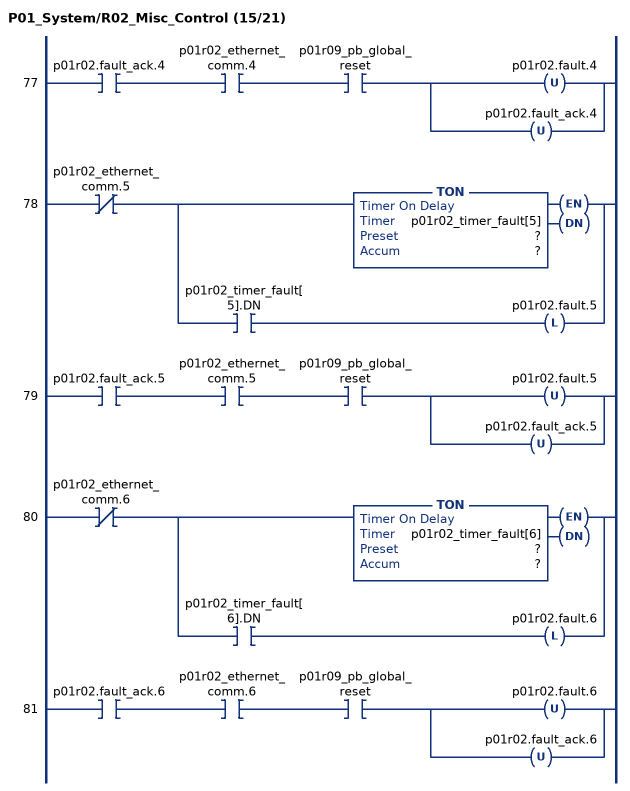
   77: XIC(p01r02.fault_ack.4)XIC(p01r02_ethernet_comm.4)XIC(p01r09_pb_global_reset)[OTU(p01r02.fault.4) ,OTU(p01r02.fault_ack.4) ];
   78: XIO(p01r02_ethernet_comm.5)[TON(p01r02_timer_fault[5],?,?) ,XIC(p01r02_timer_fault[5].DN) OTL(p01r02.fault.5) ];
   79: XIC(p01r02.fault_ack.5)XIC(p01r02_ethernet_comm.5)XIC(p01r09_pb_global_reset)[OTU(p01r02.fault.5) ,OTU(p01r02.fault_ack.5) ];
   80: XIO(p01r02_ethernet_comm.6)[TON(p01r02_timer_fault[6],?,?) ,XIC(p01r02_timer_fault[6].DN) OTL(p01r02.fault.6) ];
   81: XIC(p01r02.fault_ack.6)XIC(p01r02_ethernet_comm.6)XIC(p01r09_pb_global_reset)[OTU(p01r02.fault.6) ,OTU(p01r02.fault_ack.6) ];
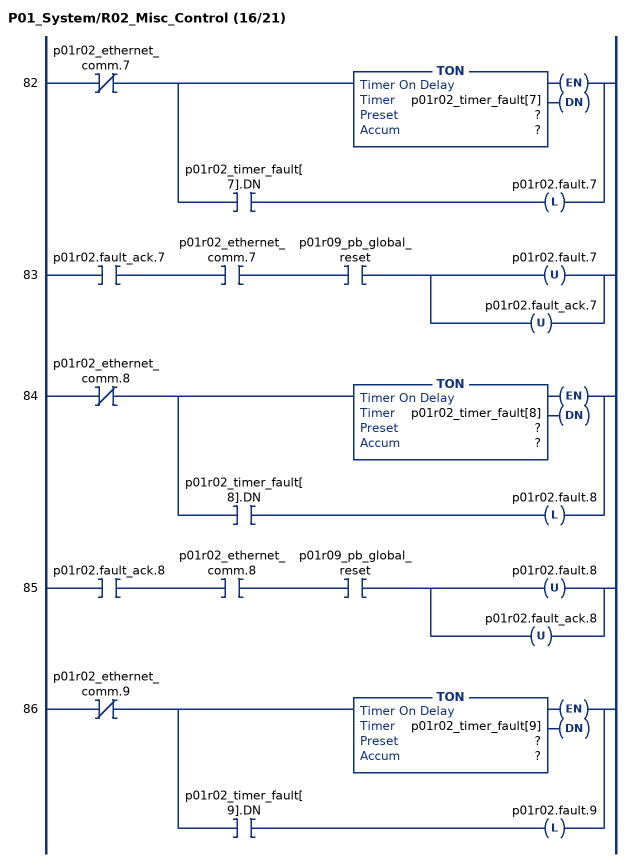
   82: XIO(p01r02_ethernet_comm.7)[TON(p01r02_timer_fault[7],?,?) ,XIC(p01r02_timer_fault[7].DN) OTL(p01r02.fault.7) ];
   83: XIC(p01r02.fault_ack.7)XIC(p01r02_ethernet_comm.7)XIC(p01r09_pb_global_reset)[OTU(p01r02.fault.7) ,OTU(p01r02.fault_ack.7) ];
   84: XIO(p01r02_ethernet_comm.8)[TON(p01r02_timer_fault[8],?,?) ,XIC(p01r02_timer_fault[8].DN) OTL(p01r02.fault.8) ];
   85: XIC(p01r02.fault_ack.8)XIC(p01r02_ethernet_comm.8)XIC(p01r09_pb_global_reset)[OTU(p01r02.fault.8) ,OTU(p01r02.fault_ack.8) ];
   86: XIO(p01r02_ethernet_comm.9)[TON(p01r02_timer_fault[9],?,?) ,XIC(p01r02_timer_fault[9].DN) OTL(p01r02.fault.9) ];
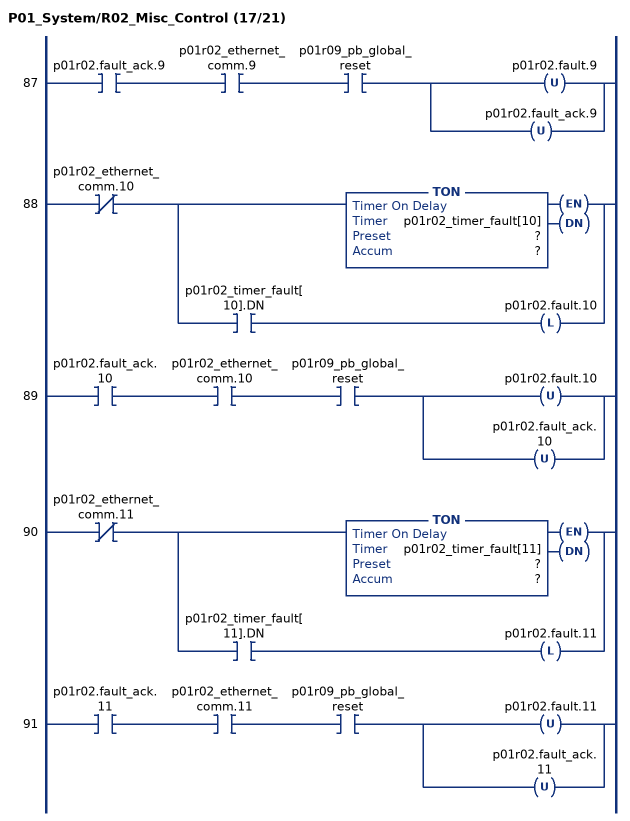
   87: XIC(p01r02.fault_ack.9)XIC(p01r02_ethernet_comm.9)XIC(p01r09_pb_global_reset)[OTU(p01r02.fault.9) ,OTU(p01r02.fault_ack.9) ];
   88: XIO(p01r02_ethernet_comm.10)[TON(p01r02_timer_fault[10],?,?) ,XIC(p01r02_timer_fault[10].DN) OTL(p01r02.fault.10) ];
   89: XIC(p01r02.fault_ack.10)XIC(p01r02_ethernet_comm.10)XIC(p01r09_pb_global_reset)[OTU(p01r02.fault.10) ,OTU(p01r02.fault_ack.10) ];
   90: XIO(p01r02_ethernet_comm.11)[TON(p01r02_timer_fault[11],?,?) ,XIC(p01r02_timer_fault[11].DN) OTL(p01r02.fault.11) ];
   91: XIC(p01r02.fault_ack.11)XIC(p01r02_ethernet_comm.11)XIC(p01r09_pb_global_reset)[OTU(p01r02.fault.11) ,OTU(p01r02.fault_ack.11) ];
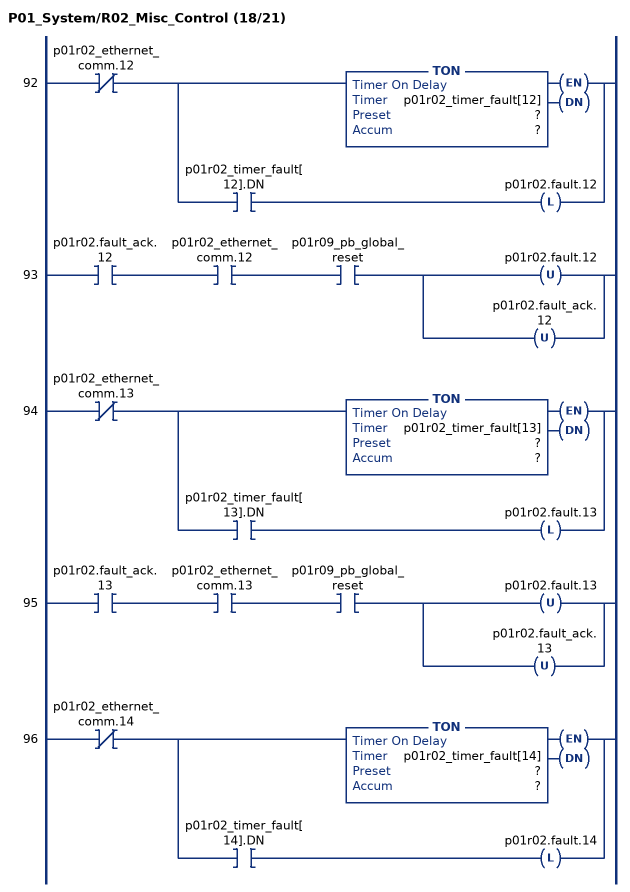
   92: XIO(p01r02_ethernet_comm.12)[TON(p01r02_timer_fault[12],?,?) ,XIC(p01r02_timer_fault[12].DN) OTL(p01r02.fault.12) ];
   93: XIC(p01r02.fault_ack.12)XIC(p01r02_ethernet_comm.12)XIC(p01r09_pb_global_reset)[OTU(p01r02.fault.12) ,OTU(p01r02.fault_ack.12) ];
   94: XIO(p01r02_ethernet_comm.13)[TON(p01r02_timer_fault[13],?,?) ,XIC(p01r02_timer_fault[13].DN) OTL(p01r02.fault.13) ];
   95: XIC(p01r02.fault_ack.13)XIC(p01r02_ethernet_comm.13)XIC(p01r09_pb_global_reset)[OTU(p01r02.fault.13) ,OTU(p01r02.fault_ack.13) ];
   96: XIO(p01r02_ethernet_comm.14)[TON(p01r02_timer_fault[14],?,?) ,XIC(p01r02_timer_fault[14].DN) OTL(p01r02.fault.14) ];
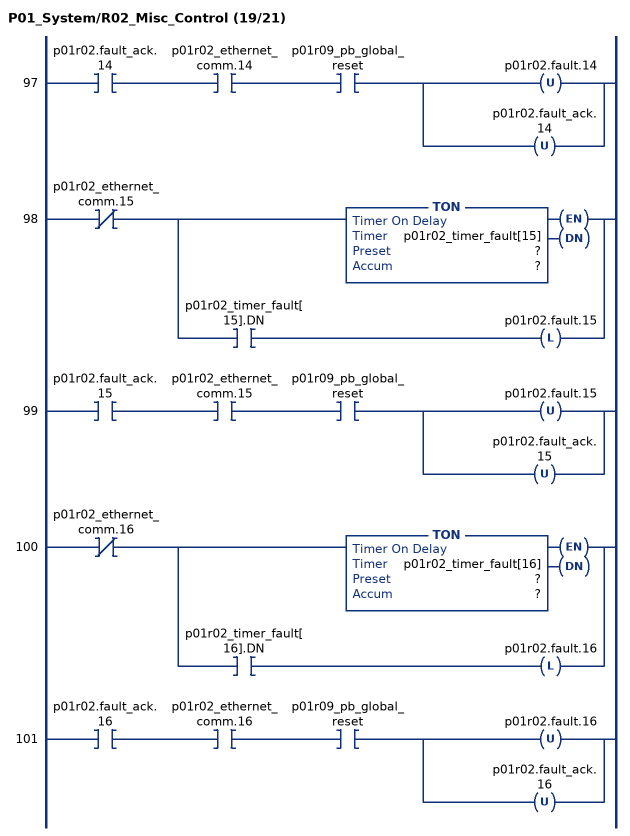
   97: XIC(p01r02.fault_ack.14)XIC(p01r02_ethernet_comm.14)XIC(p01r09_pb_global_reset)[OTU(p01r02.fault.14) ,OTU(p01r02.fault_ack.14) ];
   98: XIO(p01r02_ethernet_comm.15)[TON(p01r02_timer_fault[15],?,?) ,XIC(p01r02_timer_fault[15].DN) OTL(p01r02.fault.15) ];
   99: XIC(p01r02.fault_ack.15)XIC(p01r02_ethernet_comm.15)XIC(p01r09_pb_global_reset)[OTU(p01r02.fault.15) ,OTU(p01r02.fault_ack.15) ];
   100: XIO(p01r02_ethernet_comm.16)[TON(p01r02_timer_fault[16],?,?) ,XIC(p01r02_timer_fault[16].DN) OTL(p01r02.fault.16) ];
   101: XIC(p01r02.fault_ack.16)XIC(p01r02_ethernet_comm.16)XIC(p01r09_pb_global_reset)[OTU(p01r02.fault.16) ,OTU(p01r02.fault_ack.16) ];
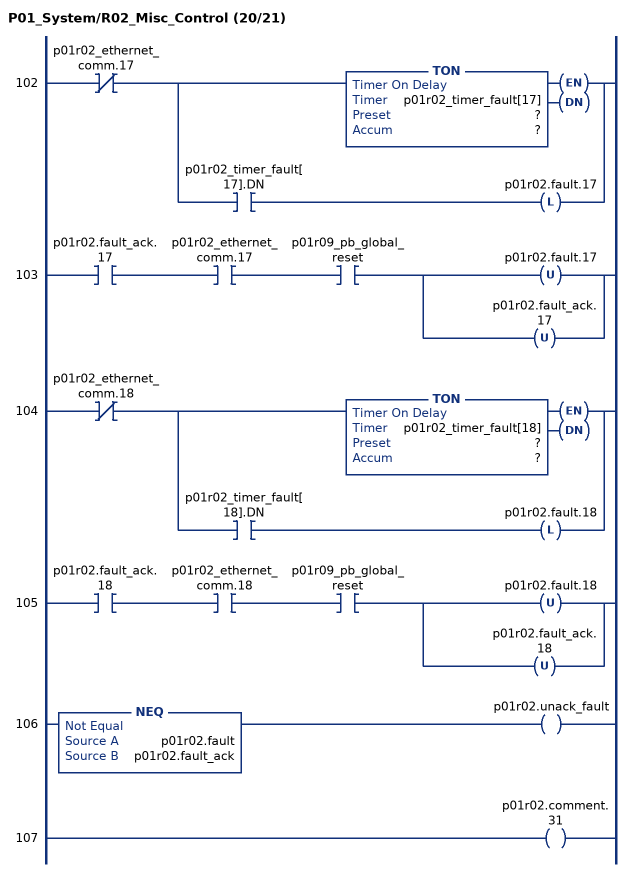
   102: XIO(p01r02_ethernet_comm.17)[TON(p01r02_timer_fault[17],?,?) ,XIC(p01r02_timer_fault[17].DN) OTL(p01r02.fault.17) ];
   103: XIC(p01r02.fault_ack.17)XIC(p01r02_ethernet_comm.17)XIC(p01r09_pb_global_reset)[OTU(p01r02.fault.17) ,OTU(p01r02.fault_ack.17) ];
   104: XIO(p01r02_ethernet_comm.18)[TON(p01r02_timer_fault[18],?,?) ,XIC(p01r02_timer_fault[18].DN) OTL(p01r02.fault.18) ];
   105: XIC(p01r02.fault_ack.18)XIC(p01r02_ethernet_comm.18)XIC(p01r09_pb_global_reset)[OTU(p01r02.fault.18) ,OTU(p01r02.fault_ack.18) ];
   106: NEQ(p01r02.fault,p01r02.fault_ack)OTE(p01r02.unack_fault);
   107: OTE(p01r02.comment.31);
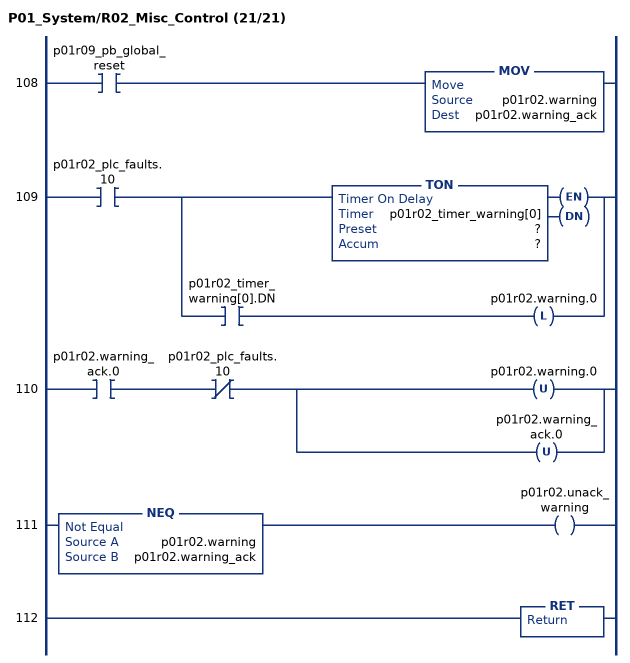
   108: XIC(p01r09_pb_global_reset)MOV(p01r02.warning,p01r02.warning_ack);
   109: XIC(p01r02_plc_faults.10)[TON(p01r02_timer_warning[0],?,?) ,XIC(p01r02_timer_warning[0].DN) OTL(p01r02.warning.0) ];
   110: XIC(p01r02.warning_ack.0)XIO(p01r02_plc_faults.10)[OTU(p01r02.warning.0) ,OTU(p01r02.warning_ack.0) ];
   111: NEQ(p01r02.warning,p01r02.warning_ack)OTE(p01r02.unack_warning);
   112: RET();
END_ROUTINE
